C01800=1075.435,113.912,-70.031,173.707,24.375,154.288
C01801=1075.430,113.662,-70.011,173.705,24.372,154.287
C01802=1075.424,113.413,-69.992,173.704,24.370,154.287
C01803=1075.418,113.163,-69.973,173.702,24.367,154.287
C01804=1075.413,112.915,-69.954,173.700,24.364,154.287
C01805=1075.407,112.666,-69.935,173.699,24.362,154.286
C01806=1075.401,112.416,-69.916,173.697,24.360,154.286
C01807=1075.395,112.167,-69.896,173.695,24.357,154.286
C01808=1075.389,111.918,-69.877,173.694,24.355,154.285
C01809=1075.384,111.669,-69.858,173.693,24.352,154.285
C01810=1075.378,111.387,-69.837,173.690,24.349,154.285
C01811=1075.371,111.105,-69.815,173.688,24.346,154.284
C01812=1075.364,110.824,-69.794,173.687,24.343,154.284
C01813=1075.358,110.542,-69.773,173.684,24.341,154.284
C01814=1075.352,110.293,-69.754,173.683,24.338,154.283
C01815=1075.347,110.044,-69.734,173.681,24.335,154.283
C01816=1075.341,109.795,-69.716,173.680,24.333,154.283
C01817=1075.335,109.546,-69.697,173.678,24.330,154.283
C01818=1075.329,109.296,-69.678,173.676,24.328,154.282
C01819=1075.323,109.047,-69.659,173.675,24.325,154.282
C01820=1075.317,108.798,-69.640,173.673,24.323,154.282
C01821=1075.312,108.549,-69.621,173.671,24.320,154.282
C01822=1075.306,108.300,-69.602,173.670,24.318,154.281
C01823=1075.300,108.050,-69.583,173.668,24.316,154.281
C01824=1075.294,107.801,-69.564,173.666,24.313,154.281
C01825=1075.289,107.552,-69.545,173.665,24.311,154.280
C01826=1075.283,107.302,-69.527,173.663,24.308,154.280
C01827=1075.277,107.053,-69.508,173.661,24.305,154.280
C01828=1075.272,106.804,-69.489,173.660,24.303,154.279
C01829=1075.266,106.555,-69.470,173.658,24.300,154.279
C01830=1075.260,106.306,-69.451,173.656,24.298,154.279
C01831=1075.255,106.056,-69.432,173.655,24.295,154.279
C01832=1075.249,105.808,-69.413,173.653,24.293,154.278
C01833=1075.243,105.558,-69.395,173.651,24.290,154.278
C01834=1075.237,105.309,-69.376,173.650,24.287,154.278
C01835=1075.232,105.060,-69.357,173.649,24.285,154.277
C01836=1075.226,104.811,-69.338,173.646,24.282,154.277
C01837=1075.220,104.561,-69.320,173.645,24.280,154.277
C01838=1075.215,104.312,-69.301,173.644,24.277,154.277
C01839=1075.209,104.063,-69.282,173.642,24.275,154.276
C01840=1075.203,103.814,-69.263,173.640,24.272,154.276
C01841=1075.198,103.565,-69.244,173.639,24.269,154.276
C01842=1075.192,103.315,-69.226,173.637,24.267,154.275
C01843=1075.186,103.066,-69.207,173.635,24.264,154.275
C01844=1075.181,102.817,-69.188,173.634,24.262,154.275
C01845=1075.175,102.567,-69.170,173.632,24.260,154.274
C01846=1075.169,102.318,-69.151,173.630,24.256,154.274
C01847=1075.164,102.069,-69.132,173.629,24.254,154.274
C01848=1075.158,101.820,-69.114,173.627,24.252,154.274
C01849=1075.153,101.571,-69.096,173.625,24.249,154.273
C01850=1075.146,101.321,-69.077,173.624,24.247,154.273
C01851=1075.141,101.071,-69.058,173.623,24.244,154.273
C01852=1075.135,100.823,-69.040,173.621,24.241,154.272
C01853=1075.129,100.574,-69.021,173.619,24.239,154.272
C01854=1075.123,100.324,-69.003,173.618,24.236,154.272
C01855=1075.118,100.075,-68.984,173.616,24.234,154.271
C01856=1075.112,99.826,-68.965,173.614,24.231,154.271
C01857=1075.106,99.576,-68.947,173.613,24.229,154.271
C01858=1075.101,99.327,-68.929,173.611,24.227,154.271
C01859=1075.095,99.078,-68.911,173.609,24.224,154.270
C01860=1075.089,98.828,-68.891,173.608,24.221,154.270
C01861=1075.083,98.580,-68.873,173.606,24.219,154.270
C01862=1075.077,98.330,-68.855,173.605,24.216,154.269
C01863=1075.072,98.081,-68.836,173.603,24.213,154.269
C01864=1075.066,97.832,-68.818,173.602,24.211,154.269
C01865=1075.060,97.582,-68.799,173.600,24.209,154.269
C01866=1075.054,97.333,-68.782,173.598,24.206,154.268
C01867=1075.048,97.084,-68.763,173.597,24.203,154.268
C01868=1075.043,96.835,-68.745,173.595,24.201,154.268
C01869=1075.037,96.586,-68.726,173.593,24.198,154.267
C01870=1075.031,96.336,-68.708,173.592,24.196,154.267
C01871=1075.026,96.087,-68.689,173.590,24.193,154.267
C01872=1075.019,95.837,-68.671,173.589,24.191,154.266
C01873=1075.014,95.589,-68.652,173.587,24.188,154.266
C01874=1075.008,95.307,-68.632,173.586,24.185,154.266
C01875=1075.001,95.025,-68.612,173.583,24.182,154.265
C01876=1074.995,94.744,-68.591,173.582,24.180,154.265
C01877=1074.988,94.462,-68.570,173.580,24.176,154.265
C01878=1074.983,94.213,-68.551,173.579,24.174,154.264
C01879=1074.977,93.963,-68.533,173.576,24.171,154.264
C01880=1074.971,93.714,-68.516,173.575,24.168,154.264
C01881=1074.965,93.465,-68.497,173.574,24.166,154.263
C01882=1074.960,93.216,-68.479,173.572,24.164,154.263
C01883=1074.953,92.967,-68.460,173.570,24.161,154.263
C01884=1074.949,92.717,-68.442,173.569,24.159,154.263
C01885=1074.943,92.468,-68.424,173.568,24.156,154.262
C01886=1074.937,92.219,-68.406,173.566,24.153,154.262
C01887=1074.931,91.970,-68.388,173.564,24.151,154.262
C01888=1074.926,91.720,-68.370,173.563,24.148,154.261
C01889=1074.919,91.471,-68.351,173.561,24.145,154.261
C01890=1074.914,91.222,-68.334,173.559,24.143,154.261
C01891=1074.909,90.972,-68.315,173.558,24.140,154.260
C01892=1074.903,90.724,-68.297,173.556,24.138,154.260
C01893=1074.897,90.474,-68.279,173.555,24.136,154.260
C01894=1074.891,90.225,-68.261,173.553,24.132,154.259
C01895=1074.885,89.975,-68.243,173.552,24.130,154.259
C01896=1074.879,89.727,-68.225,173.550,24.128,154.259
C01897=1074.874,89.477,-68.207,173.549,24.125,154.259
C01898=1074.868,89.228,-68.189,173.547,24.122,154.258
C01899=1074.862,88.978,-68.171,173.545,24.120,154.258
C01900=1074.856,88.729,-68.153,173.544,24.117,154.258
C01901=1074.850,88.480,-68.135,173.543,24.115,154.257
C01902=1074.844,88.230,-68.117,173.541,24.112,154.257
C01903=1074.839,87.981,-68.099,173.539,24.110,154.257
C01904=1074.833,87.732,-68.081,173.538,24.107,154.257
C01905=1074.827,87.483,-68.063,173.537,24.105,154.256
C01906=1074.821,87.234,-68.046,173.534,24.102,154.256
C01907=1074.815,86.984,-68.028,173.533,24.099,154.256
C01908=1074.810,86.735,-68.010,173.532,24.097,154.255
C01909=1074.804,86.485,-67.992,173.530,24.095,154.255
C01910=1074.798,86.236,-67.973,173.528,24.092,154.255
C01911=1074.792,85.987,-67.955,173.527,24.089,154.254
C01912=1074.787,85.738,-67.938,173.526,24.087,154.254
C01913=1074.780,85.488,-67.920,173.524,24.084,154.254
C01914=1074.775,85.239,-67.902,173.522,24.081,154.254
C01915=1074.769,84.989,-67.884,173.521,24.079,154.253
C01916=1074.763,84.740,-67.867,173.519,24.076,154.253
C01917=1074.758,84.491,-67.849,173.518,24.074,154.253
C01918=1074.752,84.241,-67.831,173.516,24.071,154.252
C01919=1074.746,83.992,-67.814,173.514,24.069,154.252
C01920=1074.740,83.743,-67.795,173.513,24.066,154.252
C01921=1074.734,83.494,-67.778,173.512,24.063,154.251
C01922=1074.729,83.245,-67.760,173.510,24.061,154.251
C01923=1074.723,82.995,-67.742,173.508,24.058,154.251
C01924=1074.717,82.746,-67.725,173.507,24.056,154.250
C01925=1074.711,82.497,-67.707,173.506,24.053,154.250
C01926=1074.705,82.247,-67.689,173.504,24.050,154.250
C01927=1074.700,81.998,-67.671,173.502,24.048,154.249
C01928=1074.694,81.749,-67.654,173.501,24.046,154.249
C01929=1074.688,81.500,-67.636,173.500,24.043,154.249
C01930=1074.683,81.251,-67.618,173.497,24.040,154.249
C01931=1074.677,81.001,-67.600,173.496,24.038,154.248
C01932=1074.671,80.752,-67.583,173.495,24.035,154.248
C01933=1074.666,80.503,-67.565,173.494,24.032,154.248
C01934=1074.659,80.253,-67.547,173.491,24.030,154.247
C01935=1074.654,80.003,-67.531,173.490,24.027,154.247
C01936=1074.649,79.754,-67.513,173.489,24.024,154.247
C01937=1074.643,79.505,-67.495,173.487,24.022,154.246
C01938=1074.636,79.224,-67.475,173.485,24.019,154.246
C01939=1074.630,78.942,-67.455,173.484,24.016,154.246
C01940=1074.624,78.661,-67.435,173.482,24.013,154.245
C01941=1074.617,78.379,-67.415,173.481,24.010,154.245
C01942=1074.612,78.129,-67.398,173.478,24.007,154.245
C01943=1074.606,77.880,-67.380,173.477,24.005,154.244
C01944=1074.600,77.631,-67.363,173.476,24.003,154.244
C01945=1074.594,77.382,-67.346,173.475,24.000,154.244
C01946=1074.588,77.132,-67.328,173.472,23.997,154.243
C01947=1074.582,76.883,-67.310,173.471,23.994,154.243
C01948=1074.577,76.634,-67.292,173.470,23.992,154.243
C01949=1074.571,76.384,-67.275,173.469,23.989,154.242
C01950=1074.564,76.135,-67.258,173.467,23.987,154.242
C01951=1074.559,75.886,-67.241,173.465,23.984,154.242
C01952=1074.553,75.637,-67.223,173.464,23.982,154.242
C01953=1074.547,75.387,-67.205,173.462,23.979,154.241
C01954=1074.542,75.137,-67.188,173.461,23.976,154.241
C01955=1074.536,74.889,-67.171,173.459,23.974,154.241
C01956=1074.530,74.639,-67.153,173.457,23.971,154.240
C01957=1074.524,74.390,-67.136,173.456,23.969,154.240
C01958=1074.519,74.140,-67.119,173.455,23.966,154.240
C01959=1074.512,73.891,-67.102,173.454,23.964,154.239
C01960=1074.507,73.642,-67.084,173.451,23.961,154.239
C01961=1074.501,73.392,-67.067,173.450,23.958,154.239
C01962=1074.496,73.143,-67.050,173.449,23.956,154.238
C01963=1074.489,72.894,-67.032,173.448,23.953,154.238
C01964=1074.483,72.645,-67.015,173.446,23.951,154.238
C01965=1074.478,72.395,-66.998,173.444,23.948,154.237
C01966=1074.473,72.146,-66.980,173.443,23.945,154.237
C01967=1074.466,71.897,-66.963,173.441,23.943,154.237
C01968=1074.461,71.647,-66.946,173.440,23.940,154.237
C01969=1074.455,71.398,-66.929,173.438,23.937,154.236
C01970=1074.449,71.149,-66.912,173.437,23.935,154.236
C01971=1074.443,70.899,-66.894,173.435,23.932,154.236
C01972=1074.438,70.650,-66.877,173.434,23.930,154.235
C01973=1074.432,70.400,-66.860,173.433,23.927,154.235
C01974=1074.426,70.151,-66.843,173.431,23.924,154.235
C01975=1074.420,69.902,-66.825,173.429,23.922,154.234
C01976=1074.414,69.652,-66.809,173.428,23.919,154.234
C01977=1074.408,69.403,-66.791,173.427,23.917,154.234
C01978=1074.403,69.154,-66.774,173.425,23.914,154.233
C01979=1074.396,68.904,-66.757,173.423,23.911,154.233
C01980=1074.391,68.655,-66.740,173.422,23.909,154.233
C01981=1074.386,68.405,-66.723,173.421,23.906,154.232
C01982=1074.379,68.157,-66.706,173.419,23.904,154.232
C01983=1074.374,67.907,-66.689,173.418,23.901,154.232
C01984=1074.367,67.658,-66.672,173.416,23.898,154.231
C01985=1074.362,67.408,-66.655,173.415,23.896,154.231
C01986=1074.356,67.159,-66.638,173.413,23.893,154.231
C01987=1074.351,66.910,-66.621,173.412,23.891,154.231
C01988=1074.345,66.660,-66.603,173.411,23.888,154.230
C01989=1074.339,66.410,-66.587,173.408,23.885,154.230
C01990=1074.333,66.161,-66.569,173.407,23.883,154.230
C01991=1074.327,65.912,-66.553,173.406,23.881,154.229
C01992=1074.322,65.663,-66.535,173.405,23.878,154.229
C01993=1074.316,65.414,-66.519,173.403,23.875,154.229
C01994=1074.310,65.163,-66.502,173.401,23.872,154.228
C01995=1074.304,64.915,-66.485,173.400,23.870,154.228
C01996=1074.298,64.665,-66.468,173.399,23.867,154.228
C01997=1074.292,64.416,-66.451,173.397,23.865,154.227
C01998=1074.287,64.167,-66.434,173.396,23.862,154.227
C01999=1074.281,63.918,-66.417,173.394,23.860,154.227
C02000=1074.274,63.668,-66.401,173.392,23.857,154.226
C02001=1074.269,63.418,-66.384,173.391,23.854,154.226
C02002=1074.262,63.137,-66.365,173.389,23.852,154.226
C02003=1074.255,62.855,-66.346,173.388,23.849,154.226
C02004=1074.248,62.574,-66.327,173.386,23.846,154.225
C02005=1074.242,62.293,-66.308,173.384,23.843,154.225
C02006=1074.236,62.042,-66.291,173.383,23.841,154.225
C02007=1074.230,61.793,-66.274,173.382,23.838,154.224
C02008=1074.224,61.544,-66.258,173.380,23.835,154.224
C02009=1074.218,61.294,-66.241,173.378,23.833,154.224
C02010=1074.212,61.046,-66.224,173.377,23.830,154.223
C02011=1074.206,60.796,-66.208,173.376,23.828,154.223
C02012=1074.200,60.546,-66.191,173.374,23.825,154.223
C02013=1074.194,60.297,-66.174,173.373,23.822,154.222
C02014=1074.188,60.048,-66.157,173.371,23.820,154.222
C02015=1074.182,59.799,-66.141,173.370,23.817,154.222
C02016=1074.177,59.549,-66.124,173.368,23.815,154.222
C02017=1074.171,59.300,-66.107,173.367,23.812,154.221
C02018=1074.164,59.050,-66.091,173.366,23.810,154.221
C02019=1074.159,58.800,-66.074,173.364,23.807,154.221
C02020=1074.153,58.551,-66.058,173.362,23.804,154.220
C02021=1074.147,58.302,-66.041,173.361,23.802,154.220
C02022=1074.141,58.053,-66.024,173.360,23.799,154.220
C02023=1074.136,57.803,-66.008,173.358,23.797,154.219
C02024=1074.130,57.554,-65.991,173.357,23.794,154.219
C02025=1074.124,57.305,-65.975,173.355,23.792,154.219
C02026=1074.118,57.055,-65.959,173.354,23.789,154.218
C02027=1074.112,56.806,-65.941,173.352,23.786,154.218
C02028=1074.106,56.556,-65.925,173.351,23.784,154.218
C02029=1074.100,56.307,-65.908,173.350,23.781,154.217
C02030=1074.094,56.058,-65.892,173.348,23.778,154.217
C02031=1074.089,55.808,-65.875,173.346,23.776,154.217
C02032=1074.083,55.559,-65.859,173.345,23.773,154.217
C02033=1074.077,55.309,-65.843,173.344,23.771,154.216
C02034=1074.070,55.060,-65.826,173.342,23.768,154.216
C02035=1074.065,54.811,-65.809,173.341,23.766,154.216
C02036=1074.059,54.561,-65.793,173.339,23.763,154.215
C02037=1074.053,54.312,-65.776,173.338,23.761,154.215
C02038=1074.047,54.063,-65.760,173.336,23.758,154.215
C02039=1074.041,53.813,-65.744,173.335,23.755,154.214
C02040=1074.036,53.564,-65.727,173.334,23.753,154.214
C02041=1074.030,53.314,-65.711,173.333,23.750,154.214
C02042=1074.024,53.065,-65.695,173.330,23.747,154.213
C02043=1074.018,52.816,-65.678,173.329,23.745,154.213
C02044=1074.012,52.566,-65.662,173.328,23.742,154.213
C02045=1074.007,52.317,-65.645,173.327,23.739,154.212
C02046=1074.001,52.067,-65.629,173.325,23.737,154.212
C02047=1073.995,51.818,-65.613,173.323,23.734,154.212
C02048=1073.989,51.569,-65.596,173.322,23.731,154.211
C02049=1073.983,51.319,-65.580,173.321,23.729,154.211
C02050=1073.978,51.070,-65.563,173.319,23.727,154.211
C02051=1073.972,50.820,-65.547,173.318,23.724,154.210
C02052=1073.966,50.571,-65.531,173.317,23.721,154.210
C02053=1073.960,50.322,-65.515,173.315,23.718,154.210
C02054=1073.954,50.072,-65.498,173.313,23.716,154.210
C02055=1073.949,49.823,-65.481,173.312,23.713,154.209
C02056=1073.943,49.573,-65.465,173.311,23.711,154.209
C02057=1073.937,49.324,-65.449,173.309,23.708,154.209
C02058=1073.931,49.075,-65.433,173.308,23.705,154.208
C02059=1073.925,48.825,-65.416,173.306,23.703,154.208
C02060=1073.919,48.576,-65.400,173.305,23.700,154.208
C02061=1073.914,48.327,-65.384,173.304,23.697,154.207
C02062=1073.909,48.078,-65.367,173.302,23.695,154.207
C02063=1073.903,47.828,-65.352,173.301,23.693,154.207
C02064=1073.897,47.578,-65.336,173.300,23.690,154.206
C02065=1073.891,47.329,-65.319,173.298,23.687,154.206
C02066=1073.885,47.047,-65.301,173.296,23.684,154.206
C02067=1073.878,46.766,-65.283,173.295,23.681,154.205
C02068=1073.871,46.483,-65.264,173.293,23.678,154.205
C02069=1073.865,46.202,-65.246,173.292,23.675,154.205
C02070=1073.859,45.952,-65.230,173.291,23.673,154.204
C02071=1073.854,45.703,-65.213,173.288,23.669,154.204
C02072=1073.848,45.454,-65.197,173.287,23.667,154.204
C02073=1073.843,45.204,-65.182,173.286,23.664,154.203
C02074=1073.837,44.955,-65.165,173.285,23.662,154.203
C02075=1073.831,44.705,-65.149,173.283,23.659,154.203
C02076=1073.825,44.456,-65.133,173.282,23.656,154.202
C02077=1073.819,44.206,-65.117,173.280,23.654,154.202
C02078=1073.813,43.957,-65.101,173.279,23.651,154.202
C02079=1073.808,43.708,-65.085,173.278,23.648,154.201
C02080=1073.802,43.459,-65.069,173.276,23.646,154.201
C02081=1073.796,43.209,-65.053,173.275,23.644,154.201
C02082=1073.790,42.959,-65.037,173.274,23.641,154.200
C02083=1073.785,42.710,-65.021,173.272,23.638,154.200
C02084=1073.779,42.461,-65.005,173.270,23.635,154.200
C02085=1073.773,42.211,-64.989,173.269,23.633,154.199
C02086=1073.767,41.961,-64.973,173.268,23.631,154.199
C02087=1073.761,41.712,-64.957,173.266,23.628,154.199
C02088=1073.756,41.463,-64.941,173.265,23.625,154.198
C02089=1073.750,41.213,-64.925,173.264,23.623,154.198
C02090=1073.743,40.964,-64.910,173.262,23.620,154.198
C02091=1073.738,40.714,-64.894,173.260,23.617,154.198
C02092=1073.732,40.465,-64.878,173.259,23.615,154.197
C02093=1073.726,40.216,-64.861,173.258,23.612,154.197
C02094=1073.721,39.966,-64.846,173.257,23.609,154.197
C02095=1073.715,39.717,-64.830,173.255,23.607,154.196
C02096=1073.709,39.467,-64.814,173.254,23.605,154.196
C02097=1073.703,39.218,-64.798,173.252,23.601,154.196
C02098=1073.697,38.968,-64.782,173.251,23.599,154.195
C02099=1073.691,38.719,-64.767,173.249,23.596,154.195
C02100=1073.686,38.470,-64.751,173.248,23.594,154.195
C02101=1073.680,38.220,-64.736,173.247,23.591,154.194
C02102=1073.674,37.971,-64.719,173.246,23.589,154.194
C02103=1073.668,37.721,-64.703,173.244,23.586,154.194
C02104=1073.662,37.471,-64.688,173.242,23.584,154.194
C02105=1073.656,37.222,-64.672,173.241,23.581,154.193
C02106=1073.651,36.973,-64.657,173.240,23.578,154.193
C02107=1073.645,36.724,-64.640,173.238,23.576,154.193
C02108=1073.638,36.474,-64.625,173.237,23.573,154.192
C02109=1073.632,36.225,-64.609,173.236,23.570,154.192
C02110=1073.627,35.975,-64.594,173.234,23.568,154.192
C02111=1073.621,35.726,-64.578,173.232,23.565,154.191
C02112=1073.615,35.476,-64.563,173.231,23.563,154.191
C02113=1073.609,35.227,-64.547,173.230,23.560,154.191
C02114=1073.603,34.977,-64.531,173.229,23.558,154.190
C02115=1073.597,34.728,-64.515,173.227,23.555,154.190
C02116=1073.592,34.479,-64.500,173.226,23.553,154.190
C02117=1073.586,34.229,-64.484,173.224,23.550,154.189
C02118=1073.579,33.980,-64.469,173.222,23.548,154.189
C02119=1073.574,33.730,-64.453,173.221,23.545,154.189
C02120=1073.568,33.480,-64.437,173.220,23.542,154.189
C02121=1073.562,33.232,-64.423,173.219,23.540,154.188
C02122=1073.556,32.982,-64.406,173.217,23.537,154.188
C02123=1073.550,32.732,-64.391,173.216,23.534,154.188
C02124=1073.544,32.483,-64.376,173.214,23.532,154.187
C02125=1073.539,32.234,-64.360,173.213,23.529,154.187
C02126=1073.533,31.984,-64.344,173.211,23.527,154.187
C02127=1073.526,31.735,-64.329,173.210,23.524,154.186
C02128=1073.521,31.485,-64.313,173.209,23.521,154.186
C02129=1073.516,31.236,-64.298,173.208,23.519,154.186
C02130=1073.508,30.954,-64.281,173.206,23.516,154.185
C02131=1073.502,30.672,-64.263,173.204,23.513,154.185
C02132=1073.495,30.390,-64.246,173.203,23.510,154.185
C02133=1073.489,30.108,-64.228,173.201,23.507,154.184
C02134=1073.483,29.859,-64.213,173.200,23.505,154.184
C02135=1073.477,29.609,-64.197,173.199,23.502,154.184
C02136=1073.471,29.360,-64.182,173.197,23.499,154.183
C02137=1073.465,29.110,-64.167,173.196,23.497,154.183
C02138=1073.459,28.861,-64.150,173.194,23.494,154.183
C02139=1073.453,28.612,-64.136,173.193,23.492,154.182
C02140=1073.448,28.362,-64.120,173.191,23.489,154.182
C02141=1073.441,28.112,-64.105,173.190,23.486,154.182
C02142=1073.436,27.864,-64.089,173.189,23.484,154.182
C02143=1073.430,27.614,-64.074,173.188,23.482,154.181
C02144=1073.424,27.364,-64.059,173.186,23.479,154.181
C02145=1073.418,27.115,-64.044,173.185,23.477,154.181
C02146=1073.413,26.865,-64.029,173.183,23.473,154.180
C02147=1073.406,26.616,-64.013,173.182,23.471,154.180
C02148=1073.400,26.366,-63.998,173.180,23.469,154.180
C02149=1073.394,26.117,-63.983,173.179,23.466,154.179
C02150=1073.389,25.867,-63.967,173.178,23.464,154.179
C02151=1073.382,25.618,-63.953,173.176,23.461,154.179
C02152=1073.376,25.369,-63.937,173.175,23.458,154.178
C02153=1073.371,25.119,-63.922,173.173,23.456,154.178
C02154=1073.364,24.870,-63.907,173.172,23.453,154.178
C02155=1073.359,24.620,-63.892,173.170,23.451,154.178
C02156=1073.353,24.371,-63.877,173.169,23.448,154.177
C02157=1073.347,24.121,-63.861,173.168,23.445,154.177
C02158=1073.342,23.872,-63.847,173.167,23.443,154.177
C02159=1073.335,23.623,-63.831,173.165,23.441,154.176
C02160=1073.329,23.373,-63.815,173.164,23.438,154.176
C02161=1073.323,23.124,-63.801,173.162,23.435,154.176
C02162=1073.318,22.874,-63.785,173.161,23.433,154.176
C02163=1073.311,22.624,-63.770,173.159,23.430,154.175
C02164=1073.306,22.375,-63.755,173.158,23.428,154.175
C02165=1073.300,22.125,-63.740,173.157,23.425,154.175
C02166=1073.294,21.876,-63.726,173.156,23.423,154.174
C02167=1073.289,21.626,-63.710,173.154,23.420,154.174
C02168=1073.282,21.377,-63.695,173.153,23.417,154.174
C02169=1073.277,21.128,-63.680,173.151,23.415,154.173
C02170=1073.271,20.878,-63.665,173.150,23.412,154.173
C02171=1073.264,20.628,-63.650,173.148,23.410,154.173
C02172=1073.259,20.379,-63.635,173.147,23.407,154.172
C02173=1073.253,20.129,-63.620,173.146,23.404,154.172
C02174=1073.247,19.880,-63.605,173.145,23.402,154.172
C02175=1073.241,19.630,-63.590,173.143,23.400,154.172
C02176=1073.235,19.381,-63.575,173.142,23.397,154.171
C02177=1073.229,19.132,-63.560,173.140,23.394,154.171
C02178=1073.223,18.882,-63.545,173.138,23.392,154.171
C02179=1073.218,18.633,-63.530,173.137,23.390,154.170
C02180=1073.211,18.383,-63.515,173.136,23.387,154.170
C02181=1073.205,18.134,-63.500,173.135,23.384,154.170
C02182=1073.200,17.884,-63.485,173.133,23.382,154.169
C02183=1073.194,17.635,-63.470,173.132,23.379,154.169
C02184=1073.188,17.386,-63.456,173.131,23.377,154.169
C02185=1073.182,17.136,-63.441,173.129,23.374,154.169
C02186=1073.176,16.887,-63.425,173.127,23.372,154.168
C02187=1073.170,16.637,-63.410,173.126,23.369,154.168
C02188=1073.165,16.387,-63.397,173.125,23.366,154.168
C02189=1073.158,16.138,-63.382,173.124,23.364,154.167
C02190=1073.153,15.888,-63.366,173.122,23.362,154.167
C02191=1073.147,15.639,-63.352,173.121,23.359,154.167
C02192=1073.140,15.389,-63.337,173.120,23.357,154.167
C02193=1073.135,15.140,-63.322,173.118,23.353,154.166
C02194=1073.128,14.860,-63.305,173.116,23.351,154.166
C02195=1073.121,14.580,-63.289,173.115,23.348,154.165
C02196=1073.115,14.299,-63.272,173.113,23.345,154.165
C02197=1073.108,14.018,-63.255,173.112,23.342,154.165
C02198=1073.102,13.769,-63.241,173.111,23.340,154.165
C02199=1073.096,13.519,-63.227,173.109,23.337,154.164
C02200=1073.090,13.270,-63.212,173.108,23.335,154.164
C02201=1073.084,13.021,-63.197,173.106,23.332,154.164
C02202=1073.078,12.770,-63.182,173.105,23.330,154.163
C02203=1073.073,12.521,-63.168,173.103,23.327,154.163
C02204=1073.066,12.271,-63.153,173.102,23.325,154.163
C02205=1073.060,12.022,-63.138,173.101,23.323,154.163
C02206=1073.054,11.772,-63.124,173.099,23.320,154.162
C02207=1073.049,11.523,-63.109,173.098,23.318,154.162
C02208=1073.042,11.274,-63.094,173.097,23.315,154.162
C02209=1073.036,11.025,-63.080,173.096,23.313,154.161
C02210=1073.030,10.774,-63.066,173.093,23.310,154.161
C02211=1073.025,10.525,-63.051,173.092,23.308,154.161
C02212=1073.018,10.276,-63.036,173.091,23.305,154.161
C02213=1073.013,10.026,-63.022,173.090,23.303,154.160
C02214=1073.006,9.776,-63.007,173.088,23.300,154.160
C02215=1073.001,9.528,-62.993,173.087,23.298,154.160
C02216=1072.994,9.277,-62.978,173.086,23.296,154.159
C02217=1072.989,9.028,-62.964,173.084,23.293,154.159
C02218=1072.982,8.779,-62.949,173.082,23.290,154.159
C02219=1072.977,8.529,-62.935,173.081,23.287,154.159
C02220=1072.970,8.279,-62.920,173.080,23.285,154.158
C02221=1072.965,8.030,-62.905,173.078,23.283,154.158
C02222=1072.959,7.780,-62.891,173.077,23.280,154.158
C02223=1072.953,7.531,-62.877,173.076,23.278,154.157
C02224=1072.946,7.282,-62.862,173.075,23.275,154.157
C02225=1072.941,7.032,-62.848,173.073,23.273,154.157
C02226=1072.935,6.782,-62.833,173.072,23.270,154.157
C02227=1072.929,6.533,-62.819,173.070,23.268,154.156
C02228=1072.923,6.283,-62.804,173.069,23.265,154.156
C02229=1072.917,6.034,-62.790,173.067,23.263,154.156
C02230=1072.911,5.785,-62.776,173.066,23.260,154.155
C02231=1072.905,5.535,-62.761,173.065,23.258,154.155
C02232=1072.900,5.285,-62.747,173.063,23.255,154.155
C02233=1072.893,5.036,-62.732,173.062,23.253,154.155
C02234=1072.888,4.786,-62.718,173.061,23.251,154.154
C02235=1072.881,4.537,-62.704,173.059,23.248,154.154
C02236=1072.875,4.287,-62.690,173.057,23.245,154.154
C02237=1072.869,4.038,-62.675,173.056,23.242,154.153
C02238=1072.863,3.788,-62.661,173.055,23.240,154.153
C02239=1072.857,3.539,-62.646,173.054,23.238,154.153
C02240=1072.852,3.289,-62.633,173.052,23.235,154.153
C02241=1072.846,3.040,-62.618,173.051,23.233,154.152
C02242=1072.840,2.790,-62.604,173.050,23.230,154.152
C02243=1072.834,2.541,-62.589,173.049,23.228,154.152
C02244=1072.828,2.291,-62.575,173.046,23.225,154.151
C02245=1072.823,2.041,-62.561,173.045,23.223,154.151
C02246=1072.816,1.792,-62.546,173.044,23.220,154.151
C02247=1072.811,1.542,-62.532,173.042,23.218,154.151
C02248=1072.805,1.293,-62.518,173.041,23.215,154.150
C02249=1072.798,1.043,-62.504,173.040,23.213,154.150
C02250=1072.793,0.794,-62.489,173.039,23.211,154.150
C02251=1072.787,0.545,-62.476,173.037,23.208,154.149
C02252=1072.781,0.294,-62.461,173.036,23.206,154.149
C02253=1072.775,0.045,-62.447,173.034,23.203,154.149
C02254=1072.770,-0.204,-62.433,173.033,23.200,154.149
C02255=1072.764,-0.454,-62.419,173.031,23.198,154.148
C02256=1072.758,-0.703,-62.404,173.030,23.196,154.148
C02257=1072.752,-0.953,-62.390,173.029,23.193,154.148
C02258=1072.745,-1.231,-62.374,173.028,23.190,154.147
C02259=1072.739,-1.510,-62.359,173.025,23.187,154.147
C02260=1072.732,-1.788,-62.343,173.024,23.184,154.147
C02261=1072.726,-2.067,-62.327,173.023,23.182,154.146
C02262=1072.720,-2.316,-62.313,173.021,23.179,154.146
C02263=1072.714,-2.565,-62.299,173.020,23.177,154.146
C02264=1072.709,-2.815,-62.285,173.018,23.174,154.146
C02265=1072.702,-3.065,-62.270,173.017,23.172,154.145
C02266=1072.697,-3.314,-62.257,173.016,23.170,154.145
C02267=1072.691,-3.564,-62.243,173.014,23.167,154.145
C02268=1072.685,-3.814,-62.229,173.013,23.165,154.145
C02269=1072.679,-4.063,-62.215,173.012,23.162,154.144
C02270=1072.673,-4.312,-62.201,173.011,23.160,154.144
C02271=1072.667,-4.562,-62.187,173.009,23.157,154.144
C02272=1072.661,-4.812,-62.173,173.007,23.155,154.143
C02273=1072.655,-5.061,-62.159,173.006,23.152,154.143
C02274=1072.648,-5.311,-62.145,173.004,23.150,154.143
C02275=1072.643,-5.560,-62.131,173.003,23.148,154.143
C02276=1072.637,-5.810,-62.118,173.002,23.145,154.142
C02277=1072.631,-6.060,-62.104,173.001,23.143,154.142
C02278=1072.625,-6.309,-62.089,172.999,23.141,154.142
C02279=1072.619,-6.558,-62.076,172.998,23.138,154.142
C02280=1072.613,-6.808,-62.062,172.997,23.136,154.141
C02281=1072.606,-7.058,-62.048,172.995,23.133,154.141
C02282=1072.601,-7.307,-62.034,172.993,23.130,154.141
C02283=1072.595,-7.557,-62.020,172.992,23.129,154.141
C02284=1072.588,-7.806,-62.006,172.991,23.126,154.140
C02285=1072.583,-8.056,-61.992,172.989,23.124,154.140
C02286=1072.577,-8.305,-61.979,172.988,23.121,154.140
C02287=1072.571,-8.555,-61.965,172.987,23.119,154.140
C02288=1072.565,-8.805,-61.951,172.985,23.116,154.139
C02289=1072.559,-9.054,-61.938,172.984,23.114,154.139
C02290=1072.553,-9.304,-61.924,172.982,23.111,154.139
C02291=1072.547,-9.553,-61.911,172.981,23.109,154.138
C02292=1072.541,-9.803,-61.896,172.979,23.107,154.138
C02293=1072.535,-10.053,-61.883,172.978,23.104,154.138
C02294=1072.529,-10.302,-61.869,172.977,23.102,154.138
C02295=1072.524,-10.551,-61.855,172.975,23.100,154.137
C02296=1072.517,-10.800,-61.841,172.974,23.097,154.137
C02297=1072.511,-11.051,-61.827,172.973,23.095,154.137
C02298=1072.505,-11.300,-61.814,172.972,23.092,154.137
C02299=1072.500,-11.549,-61.800,172.969,23.089,154.136
C02300=1072.493,-11.799,-61.787,172.968,23.088,154.136
C02301=1072.488,-12.048,-61.773,172.967,23.085,154.136
C02302=1072.481,-12.298,-61.759,172.965,23.083,154.136
C02303=1072.476,-12.548,-61.745,172.964,23.080,154.135
C02304=1072.470,-12.797,-61.731,172.963,23.078,154.135
C02305=1072.464,-13.047,-61.718,172.962,23.075,154.135
C02306=1072.458,-13.296,-61.704,172.960,23.073,154.135
C02307=1072.452,-13.545,-61.691,172.959,23.071,154.134
C02308=1072.446,-13.796,-61.677,172.958,23.069,154.134
C02309=1072.440,-14.045,-61.664,172.955,23.066,154.134
C02310=1072.435,-14.295,-61.650,172.954,23.063,154.134
C02311=1072.429,-14.544,-61.637,172.953,23.061,154.133
C02312=1072.423,-14.794,-61.623,172.952,23.059,154.133
C02313=1072.417,-15.043,-61.610,172.950,23.056,154.133
C02314=1072.411,-15.293,-61.596,172.949,23.054,154.133
C02315=1072.405,-15.543,-61.582,172.948,23.052,154.132
C02316=1072.398,-15.792,-61.569,172.946,23.049,154.132
C02317=1072.393,-16.042,-61.555,172.945,23.047,154.132
C02318=1072.387,-16.291,-61.542,172.944,23.045,154.132
C02319=1072.380,-16.540,-61.529,172.941,23.042,154.131
C02320=1072.374,-16.791,-61.515,172.940,23.040,154.131
C02321=1072.369,-17.040,-61.502,172.939,23.037,154.131
C02322=1072.362,-17.317,-61.488,172.938,23.035,154.130
C02323=1072.355,-17.594,-61.472,172.936,23.032,154.130
C02324=1072.349,-17.871,-61.458,172.934,23.030,154.130
C02325=1072.342,-18.148,-61.443,172.933,23.027,154.130
C02326=1072.336,-18.397,-61.429,172.932,23.025,154.130
C02327=1072.330,-18.646,-61.416,172.930,23.023,154.129
C02328=1072.324,-18.896,-61.402,172.929,23.020,154.129
C02329=1072.318,-19.145,-61.388,172.927,23.018,154.129
C02330=1072.312,-19.395,-61.376,172.925,23.016,154.129
C02331=1072.306,-19.644,-61.363,172.924,23.013,154.128
C02332=1072.301,-19.894,-61.349,172.923,23.011,154.128
C02333=1072.294,-20.144,-61.335,172.922,23.008,154.128
C02334=1072.288,-20.394,-61.322,172.920,23.007,154.128
C02335=1072.282,-20.643,-61.309,172.919,23.004,154.127
C02336=1072.276,-20.893,-61.295,172.918,23.002,154.127
C02337=1072.270,-21.142,-61.282,172.916,23.000,154.127
C02338=1072.264,-21.392,-61.270,172.915,22.997,154.127
C02339=1072.259,-21.641,-61.256,172.913,22.995,154.126
C02340=1072.252,-21.891,-61.242,172.911,22.992,154.126
C02341=1072.246,-22.141,-61.230,172.910,22.990,154.126
C02342=1072.240,-22.390,-61.217,172.909,22.988,154.126
C02343=1072.235,-22.639,-61.203,172.907,22.985,154.125
C02344=1072.229,-22.889,-61.189,172.906,22.983,154.125
C02345=1072.222,-23.139,-61.177,172.905,22.981,154.125
C02346=1072.216,-23.389,-61.163,172.903,22.979,154.125
C02347=1072.210,-23.638,-61.149,172.902,22.976,154.124
C02348=1072.204,-23.888,-61.137,172.901,22.974,154.124
C02349=1072.198,-24.137,-61.124,172.899,22.971,154.124
C02350=1072.192,-24.387,-61.111,172.897,22.969,154.124
C02351=1072.187,-24.637,-61.097,172.896,22.967,154.124
C02352=1072.181,-24.886,-61.084,172.895,22.965,154.123
C02353=1072.175,-25.136,-61.071,172.893,22.962,154.123
C02354=1072.168,-25.385,-61.058,172.892,22.960,154.123
C02355=1072.163,-25.635,-61.044,172.891,22.958,154.123
C02356=1072.157,-25.885,-61.032,172.889,22.955,154.122
C02357=1072.151,-26.134,-61.018,172.888,22.954,154.122
C02358=1072.145,-26.384,-61.006,172.887,22.951,154.122
C02359=1072.140,-26.633,-60.992,172.884,22.948,154.122
C02360=1072.134,-26.883,-60.979,172.883,22.946,154.121
C02361=1072.127,-27.132,-60.966,172.882,22.944,154.121
C02362=1072.121,-27.382,-60.953,172.881,22.942,154.121
C02363=1072.115,-27.632,-60.940,172.879,22.940,154.121
C02364=1072.109,-27.881,-60.927,172.878,22.937,154.120
C02365=1072.103,-28.131,-60.914,172.876,22.935,154.120
C02366=1072.097,-28.380,-60.901,172.875,22.933,154.120
C02367=1072.091,-28.630,-60.889,172.874,22.931,154.120
C02368=1072.085,-28.879,-60.875,172.872,22.929,154.120
C02369=1072.079,-29.129,-60.863,172.870,22.926,154.119
C02370=1072.073,-29.378,-60.850,172.869,22.924,154.119
C02371=1072.067,-29.628,-60.837,172.868,22.921,154.119
C02372=1072.061,-29.877,-60.824,172.866,22.920,154.119
C02373=1072.055,-30.127,-60.811,172.865,22.917,154.118
C02374=1072.048,-30.377,-60.798,172.863,22.915,154.118
C02375=1072.043,-30.626,-60.785,172.862,22.913,154.118
C02376=1072.037,-30.876,-60.773,172.861,22.911,154.118
C02377=1072.030,-31.126,-60.760,172.859,22.908,154.118
C02378=1072.024,-31.376,-60.747,172.858,22.907,154.117
C02379=1072.018,-31.625,-60.734,172.857,22.904,154.117
C02380=1072.012,-31.875,-60.721,172.854,22.902,154.117
C02381=1072.006,-32.124,-60.708,172.853,22.899,154.117
C02382=1072.000,-32.374,-60.695,172.852,22.897,154.117
C02383=1071.994,-32.624,-60.683,172.850,22.895,154.116
C02384=1071.988,-32.873,-60.670,172.849,22.893,154.116
C02385=1071.982,-33.123,-60.657,172.848,22.891,154.116
C02386=1071.976,-33.399,-60.643,172.846,22.888,154.116
C02387=1071.970,-33.675,-60.628,172.844,22.885,154.115
C02388=1071.963,-33.950,-60.615,172.843,22.884,154.115
C02389=1071.956,-34.227,-60.600,172.842,22.881,154.115
C02390=1071.950,-34.476,-60.588,172.840,22.879,154.115
C02391=1071.944,-34.726,-60.575,172.839,22.877,154.115
C02392=1071.938,-34.976,-60.562,172.837,22.874,154.114
C02393=1071.932,-35.226,-60.549,172.835,22.872,154.114
C02394=1071.926,-35.475,-60.537,172.834,22.870,154.114
C02395=1071.921,-35.724,-60.524,172.833,22.868,154.114
C02396=1071.915,-35.974,-60.511,172.831,22.865,154.113
C02397=1071.909,-36.224,-60.499,172.830,22.863,154.113
C02398=1071.903,-36.473,-60.485,172.829,22.861,154.113
C02399=1071.897,-36.723,-60.473,172.827,22.859,154.113
C02400=1071.890,-36.972,-60.461,172.826,22.857,154.113
C02401=1071.884,-37.222,-60.448,172.824,22.855,154.112
C02402=1071.879,-37.471,-60.436,172.823,22.852,154.112
C02403=1071.873,-37.721,-60.423,172.821,22.850,154.112
C02404=1071.867,-37.971,-60.410,172.819,22.848,154.112
C02405=1071.861,-38.221,-60.398,172.818,22.846,154.112
C02406=1071.855,-38.470,-60.385,172.817,22.844,154.111
C02407=1071.849,-38.720,-60.372,172.816,22.841,154.111
C02408=1071.843,-38.970,-60.359,172.814,22.839,154.111
C02409=1071.836,-39.219,-60.348,172.813,22.837,154.111
C02410=1071.831,-39.468,-60.335,172.811,22.835,154.111
C02411=1071.825,-39.718,-60.323,172.810,22.833,154.110
C02412=1071.819,-39.967,-60.309,172.809,22.831,154.110
C02413=1071.812,-40.217,-60.298,172.807,22.829,154.110
C02414=1071.806,-40.467,-60.285,172.805,22.826,154.110
C02415=1071.800,-40.717,-60.272,172.804,22.824,154.110
C02416=1071.794,-40.967,-60.260,172.802,22.822,154.109
C02417=1071.788,-41.216,-60.248,172.801,22.820,154.109
C02418=1071.782,-41.465,-60.236,172.800,22.818,154.109
C02419=1071.776,-41.715,-60.222,172.798,22.816,154.109
C02420=1071.770,-41.965,-60.210,172.797,22.814,154.109
C02421=1071.764,-42.214,-60.198,172.795,22.812,154.108
C02422=1071.758,-42.464,-60.185,172.794,22.810,154.108
C02423=1071.752,-42.714,-60.173,172.793,22.808,154.108
C02424=1071.747,-42.963,-60.161,172.791,22.805,154.108
C02425=1071.740,-43.213,-60.149,172.789,22.803,154.108
C02426=1071.734,-43.463,-60.136,172.788,22.801,154.108
C02427=1071.728,-43.712,-60.124,172.786,22.799,154.107
C02428=1071.721,-43.962,-60.112,172.785,22.797,154.107
C02429=1071.716,-44.211,-60.099,172.783,22.795,154.107
C02430=1071.710,-44.461,-60.087,172.782,22.793,154.107
C02431=1071.704,-44.711,-60.075,172.781,22.791,154.107
C02432=1071.698,-44.961,-60.062,172.779,22.789,154.106
C02433=1071.692,-45.210,-60.050,172.778,22.787,154.106
C02434=1071.686,-45.460,-60.038,172.776,22.785,154.106
C02435=1071.680,-45.709,-60.026,172.775,22.782,154.106
C02436=1071.674,-45.959,-60.013,172.774,22.781,154.106
C02437=1071.668,-46.209,-60.001,172.771,22.778,154.106
C02438=1071.662,-46.458,-59.989,172.770,22.776,154.105
C02439=1071.656,-46.708,-59.976,172.769,22.774,154.105
C02440=1071.650,-46.958,-59.964,172.767,22.772,154.105
C02441=1071.644,-47.207,-59.952,172.766,22.770,154.105
C02442=1071.638,-47.456,-59.940,172.765,22.768,154.105
C02443=1071.632,-47.706,-59.927,172.763,22.766,154.104
C02444=1071.626,-47.956,-59.915,172.762,22.764,154.104
C02445=1071.620,-48.206,-59.903,172.760,22.762,154.104
C02446=1071.614,-48.455,-59.890,172.759,22.759,154.104
C02447=1071.608,-48.704,-59.879,172.758,22.758,154.104
C02448=1071.602,-48.954,-59.866,172.756,22.756,154.104
C02449=1071.597,-49.203,-59.854,172.755,22.754,154.103
C02450=1071.590,-49.480,-59.841,172.753,22.751,154.103
C02451=1071.582,-49.757,-59.827,172.751,22.749,154.103
C02452=1071.577,-50.033,-59.814,172.750,22.747,154.103
C02453=1071.570,-50.310,-59.801,172.748,22.744,154.103
C02454=1071.564,-50.560,-59.788,172.746,22.742,154.103
C02455=1071.558,-50.809,-59.777,172.745,22.741,154.102
C02456=1071.551,-51.058,-59.765,172.743,22.739,154.102
C02457=1071.545,-51.308,-59.752,172.742,22.736,154.102
C02458=1071.539,-51.558,-59.740,172.741,22.734,154.102
C02459=1071.533,-51.808,-59.728,172.739,22.732,154.102
C02460=1071.527,-52.057,-59.717,172.738,22.730,154.102
C02461=1071.520,-52.307,-59.705,172.736,22.729,154.101
C02462=1071.514,-52.556,-59.692,172.735,22.727,154.101
C02463=1071.508,-52.806,-59.680,172.733,22.725,154.101
C02464=1071.502,-53.056,-59.669,172.731,22.722,154.101
C02465=1071.496,-53.305,-59.657,172.730,22.721,154.101
C02466=1071.489,-53.555,-59.645,172.728,22.719,154.101
C02467=1071.483,-53.804,-59.633,172.727,22.717,154.101
C02468=1071.478,-54.054,-59.621,172.725,22.715,154.100
C02469=1071.471,-54.304,-59.609,172.724,22.713,154.100
C02470=1071.464,-54.553,-59.597,172.723,22.711,154.100
C02471=1071.459,-54.803,-59.585,172.721,22.709,154.100
C02472=1071.453,-55.053,-59.574,172.720,22.707,154.100
C02473=1071.446,-55.302,-59.562,172.718,22.705,154.100
C02474=1071.441,-55.552,-59.550,172.717,22.703,154.099
C02475=1071.434,-55.801,-59.538,172.715,22.702,154.099
C02476=1071.428,-56.051,-59.527,172.714,22.700,154.099
C02477=1071.422,-56.301,-59.514,172.713,22.698,154.099
C02478=1071.416,-56.550,-59.503,172.710,22.695,154.099
C02479=1071.410,-56.800,-59.491,172.709,22.694,154.099
C02480=1071.404,-57.050,-59.479,172.707,22.692,154.099
C02481=1071.398,-57.299,-59.467,172.706,22.690,154.098
C02482=1071.391,-57.549,-59.456,172.704,22.688,154.098
C02483=1071.385,-57.799,-59.443,172.703,22.686,154.098
C02484=1071.379,-58.048,-59.432,172.702,22.684,154.098
C02485=1071.373,-58.298,-59.421,172.700,22.682,154.098
C02486=1071.368,-58.547,-59.408,172.699,22.680,154.098
C02487=1071.361,-58.798,-59.397,172.697,22.678,154.098
C02488=1071.355,-59.047,-59.385,172.696,22.676,154.097
C02489=1071.349,-59.296,-59.374,172.694,22.675,154.097
C02490=1071.343,-59.547,-59.362,172.693,22.673,154.097
C02491=1071.336,-59.796,-59.350,172.691,22.671,154.097
C02492=1071.331,-60.046,-59.339,172.690,22.669,154.097
C02493=1071.325,-60.295,-59.326,172.688,22.667,154.097
C02494=1071.319,-60.544,-59.315,172.686,22.665,154.097
C02495=1071.312,-60.795,-59.303,172.685,22.663,154.097
C02496=1071.306,-61.044,-59.291,172.683,22.661,154.096
C02497=1071.301,-61.294,-59.280,172.682,22.660,154.096
C02498=1071.294,-61.543,-59.268,172.681,22.658,154.096
C02499=1071.288,-61.793,-59.257,172.679,22.656,154.096
C02500=1071.282,-62.043,-59.245,172.678,22.654,154.096
C02501=1071.277,-62.292,-59.234,172.676,22.652,154.096
C02502=1071.270,-62.542,-59.222,172.675,22.651,154.096
C02503=1071.264,-62.792,-59.211,172.673,22.649,154.095
C02504=1071.258,-63.041,-59.198,172.672,22.647,154.095
C02505=1071.252,-63.291,-59.187,172.670,22.645,154.095
C02506=1071.246,-63.540,-59.176,172.669,22.643,154.095
C02507=1071.240,-63.791,-59.164,172.668,22.641,154.095
C02508=1071.234,-64.040,-59.152,172.666,22.639,154.095
C02509=1071.228,-64.290,-59.141,172.664,22.637,154.095
C02510=1071.222,-64.539,-59.129,172.662,22.635,154.095
C02511=1071.216,-64.789,-59.118,172.661,22.634,154.094
C02512=1071.210,-65.038,-59.107,172.659,22.632,154.094
C02513=1071.204,-65.288,-59.095,172.658,22.630,154.094
C02514=1071.197,-65.566,-59.082,172.656,22.628,154.094
C02515=1071.190,-65.844,-59.069,172.655,22.626,154.094
C02516=1071.184,-66.121,-59.056,172.653,22.624,154.094
C02517=1071.177,-66.399,-59.044,172.651,22.622,154.094
C02518=1071.171,-66.649,-59.032,172.650,22.620,154.093
C02519=1071.165,-66.898,-59.022,172.648,22.618,154.093
C02520=1071.159,-67.148,-59.009,172.647,22.616,154.093
C02521=1071.153,-67.398,-58.998,172.646,22.614,154.093
C02522=1071.147,-67.648,-58.987,172.644,22.613,154.093
C02523=1071.141,-67.897,-58.975,172.643,22.611,154.093
C02524=1071.135,-68.147,-58.964,172.641,22.609,154.093
C02525=1071.130,-68.397,-58.953,172.640,22.607,154.093
C02526=1071.123,-68.646,-58.941,172.638,22.605,154.092
C02527=1071.117,-68.896,-58.930,172.637,22.604,154.092
C02528=1071.111,-69.146,-58.918,172.634,22.602,154.092
C02529=1071.105,-69.395,-58.907,172.633,22.600,154.092
C02530=1071.100,-69.645,-58.895,172.631,22.598,154.092
C02531=1071.094,-69.895,-58.884,172.630,22.596,154.092
C02532=1071.088,-70.144,-58.873,172.628,22.594,154.092
C02533=1071.081,-70.394,-58.861,172.627,22.593,154.092
C02534=1071.075,-70.643,-58.850,172.626,22.591,154.092
C02535=1071.069,-70.894,-58.839,172.624,22.589,154.091
C02536=1071.064,-71.143,-58.827,172.623,22.587,154.091
C02537=1071.058,-71.392,-58.816,172.621,22.585,154.091
C02538=1071.052,-71.642,-58.805,172.620,22.584,154.091
C02539=1071.046,-71.892,-58.794,172.618,22.582,154.091
C02540=1071.039,-72.142,-58.782,172.617,22.580,154.091
C02541=1071.034,-72.391,-58.771,172.615,22.578,154.091
C02542=1071.028,-72.641,-58.760,172.614,22.576,154.091
C02543=1071.022,-72.891,-58.748,172.612,22.575,154.091
C02544=1071.017,-73.141,-58.738,172.611,22.573,154.090
C02545=1071.010,-73.390,-58.726,172.609,22.571,154.090
C02546=1071.004,-73.640,-58.715,172.608,22.569,154.090
C02547=1070.998,-73.889,-58.704,172.606,22.568,154.090
C02548=1070.992,-74.139,-58.693,172.605,22.566,154.090
C02549=1070.986,-74.389,-58.682,172.603,22.564,154.090
C02550=1070.980,-74.639,-58.671,172.601,22.563,154.090
C02551=1070.974,-74.888,-58.660,172.600,22.561,154.090
C02552=1070.968,-75.137,-58.648,172.598,22.559,154.090
C02553=1070.962,-75.387,-58.637,172.597,22.557,154.090
C02554=1070.956,-75.637,-58.626,172.595,22.556,154.090
C02555=1070.950,-75.887,-58.615,172.594,22.554,154.089
C02556=1070.944,-76.137,-58.604,172.592,22.552,154.089
C02557=1070.938,-76.386,-58.593,172.591,22.551,154.089
C02558=1070.931,-76.636,-58.582,172.589,22.549,154.089
C02559=1070.925,-76.886,-58.571,172.587,22.548,154.089
C02560=1070.919,-77.136,-58.560,172.586,22.546,154.089
C02561=1070.913,-77.385,-58.549,172.584,22.544,154.089
C02562=1070.907,-77.634,-58.538,172.583,22.542,154.089
C02563=1070.901,-77.884,-58.526,172.581,22.541,154.089
C02564=1070.895,-78.134,-58.516,172.580,22.539,154.089
C02565=1070.890,-78.383,-58.505,172.578,22.538,154.089
C02566=1070.883,-78.633,-58.493,172.577,22.536,154.088
C02567=1070.877,-78.883,-58.483,172.575,22.535,154.088
C02568=1070.872,-79.132,-58.472,172.574,22.533,154.088
C02569=1070.865,-79.382,-58.461,172.572,22.531,154.088
C02570=1070.859,-79.632,-58.450,172.571,22.529,154.088
C02571=1070.853,-79.881,-58.439,172.569,22.528,154.088
C02572=1070.847,-80.131,-58.428,172.568,22.526,154.088
C02573=1070.841,-80.381,-58.417,172.566,22.525,154.088
C02574=1070.834,-80.631,-58.407,172.565,22.523,154.088
C02575=1070.828,-80.880,-58.396,172.563,22.521,154.088
C02576=1070.822,-81.130,-58.385,172.562,22.520,154.088
C02577=1070.815,-81.380,-58.374,172.560,22.519,154.088
C02578=1070.810,-81.621,-58.364,172.559,22.517,154.088
C02579=1070.804,-81.862,-58.353,172.557,22.516,154.088
C02580=1070.798,-82.103,-58.343,172.555,22.514,154.088
C02581=1070.792,-82.344,-58.332,172.554,22.512,154.087
C02582=1070.786,-82.585,-58.322,172.552,22.511,154.087
C02583=1070.780,-82.826,-58.311,172.551,22.510,154.087
C02584=1070.774,-83.068,-58.302,172.549,22.508,154.087
C02585=1070.769,-83.309,-58.291,172.548,22.506,154.087
C02586=1070.763,-83.559,-58.280,172.546,22.505,154.087
C02587=1070.756,-83.809,-58.270,172.545,22.504,154.087
C02588=1070.750,-84.058,-58.259,172.543,22.502,154.087
C02589=1070.744,-84.308,-58.248,172.542,22.500,154.087
C02590=1070.737,-84.558,-58.237,172.540,22.499,154.087
C02591=1070.731,-84.807,-58.226,172.539,22.497,154.087
C02592=1070.726,-85.057,-58.215,172.537,22.496,154.087
C02593=1070.719,-85.307,-58.205,172.535,22.494,154.087
C02594=1070.712,-85.604,-58.193,172.533,22.492,154.087
C02595=1070.705,-85.900,-58.180,172.531,22.491,154.087
C02596=1070.697,-86.198,-58.167,172.529,22.488,154.087
C02597=1070.690,-86.495,-58.155,172.527,22.487,154.087
C02598=1070.685,-86.744,-58.144,172.526,22.486,154.087
C02599=1070.677,-86.994,-58.133,172.524,22.484,154.086
C02600=1070.672,-87.243,-58.122,172.523,22.482,154.086
C02601=1070.666,-87.493,-58.113,172.521,22.481,154.086
C02602=1070.660,-87.743,-58.102,172.520,22.480,154.086
C02603=1070.653,-87.993,-58.091,172.518,22.478,154.086
C02604=1070.647,-88.242,-58.080,172.517,22.476,154.086
C02605=1070.642,-88.492,-58.070,172.515,22.475,154.086
C02606=1070.636,-88.742,-58.059,172.513,22.474,154.086
C02607=1070.629,-88.992,-58.049,172.512,22.472,154.086
C02608=1070.623,-89.241,-58.038,172.510,22.470,154.086
C02609=1070.617,-89.491,-58.028,172.509,22.469,154.086
C02610=1070.611,-89.740,-58.017,172.507,22.468,154.086
C02611=1070.605,-89.991,-58.006,172.506,22.466,154.086
C02612=1070.599,-90.240,-57.996,172.504,22.465,154.086
C02613=1070.593,-90.490,-57.986,172.503,22.463,154.086
C02614=1070.586,-90.739,-57.975,172.501,22.462,154.086
C02615=1070.581,-90.989,-57.964,172.499,22.460,154.086
C02616=1070.575,-91.239,-57.954,172.498,22.459,154.086
C02617=1070.568,-91.489,-57.944,172.496,22.458,154.086
C02618=1070.562,-91.738,-57.933,172.495,22.456,154.086
C02619=1070.556,-91.988,-57.923,172.493,22.455,154.086
C02620=1070.550,-92.237,-57.912,172.492,22.453,154.086
C02621=1070.544,-92.487,-57.901,172.490,22.452,154.086
C02622=1070.538,-92.737,-57.892,172.488,22.450,154.085
C02623=1070.532,-92.987,-57.881,172.487,22.449,154.085
C02624=1070.526,-93.237,-57.871,172.485,22.448,154.085
C02625=1070.520,-93.486,-57.860,172.484,22.446,154.085
C02626=1070.514,-93.735,-57.850,172.482,22.445,154.085
C02627=1070.508,-93.986,-57.839,172.480,22.444,154.085
C02628=1070.502,-94.236,-57.829,172.479,22.442,154.085
C02629=1070.496,-94.485,-57.819,172.477,22.440,154.085
C02630=1070.490,-94.735,-57.808,172.476,22.439,154.085
C02631=1070.484,-94.984,-57.798,172.474,22.438,154.085
C02632=1070.478,-95.234,-57.788,172.472,22.436,154.085
C02633=1070.472,-95.483,-57.777,172.471,22.435,154.085
C02634=1070.466,-95.733,-57.767,172.469,22.434,154.085
C02635=1070.459,-95.983,-57.757,172.468,22.432,154.085
C02636=1070.454,-96.233,-57.746,172.466,22.431,154.085
C02637=1070.447,-96.483,-57.736,172.464,22.429,154.085
C02638=1070.442,-96.733,-57.726,172.463,22.428,154.085
C02639=1070.436,-96.982,-57.715,172.461,22.427,154.085
C02640=1070.430,-97.232,-57.705,172.460,22.425,154.085
C02641=1070.424,-97.481,-57.695,172.458,22.424,154.085
C02642=1070.417,-97.763,-57.684,172.456,22.423,154.085
C02643=1070.409,-98.046,-57.671,172.454,22.421,154.085
C02644=1070.403,-98.328,-57.660,172.452,22.420,154.085
C02645=1070.396,-98.610,-57.649,172.451,22.418,154.085
C02646=1070.390,-98.860,-57.639,172.449,22.417,154.085
C02647=1070.384,-99.110,-57.628,172.448,22.416,154.085
C02648=1070.378,-99.360,-57.618,172.446,22.414,154.085
C02649=1070.371,-99.609,-57.608,172.444,22.413,154.085
C02650=1070.366,-99.859,-57.598,172.443,22.411,154.085
C02651=1070.359,-100.109,-57.588,172.441,22.410,154.085
C02652=1070.353,-100.358,-57.578,172.440,22.409,154.085
C02653=1070.347,-100.608,-57.567,172.438,22.407,154.085
C02654=1070.341,-100.858,-57.558,172.436,22.407,154.085
C02655=1070.335,-101.107,-57.548,172.435,22.405,154.085
C02656=1070.328,-101.357,-57.538,172.433,22.404,154.085
C02657=1070.323,-101.607,-57.528,172.431,22.403,154.085
C02658=1070.316,-101.857,-57.517,172.430,22.401,154.085
C02659=1070.310,-102.106,-57.507,172.428,22.400,154.085
C02660=1070.304,-102.357,-57.497,172.426,22.399,154.085
C02661=1070.298,-102.606,-57.487,172.425,22.398,154.085
C02662=1070.292,-102.856,-57.477,172.423,22.396,154.085
C02663=1070.286,-103.106,-57.467,172.422,22.395,154.085
C02664=1070.280,-103.355,-57.457,172.420,22.394,154.085
C02665=1070.274,-103.605,-57.447,172.418,22.393,154.085
C02666=1070.267,-103.854,-57.438,172.417,22.391,154.085
C02667=1070.262,-104.104,-57.427,172.415,22.390,154.085
C02668=1070.256,-104.354,-57.417,172.413,22.389,154.085
C02669=1070.249,-104.603,-57.408,172.412,22.388,154.085
C02670=1070.244,-104.853,-57.397,172.410,22.387,154.085
C02671=1070.237,-105.103,-57.387,172.408,22.385,154.085
C02672=1070.231,-105.353,-57.378,172.407,22.384,154.085
C02673=1070.225,-105.602,-57.368,172.405,22.383,154.085
C02674=1070.219,-105.852,-57.357,172.403,22.382,154.085
C02675=1070.213,-106.102,-57.348,172.403,22.381,154.085
C02676=1070.207,-106.351,-57.338,172.401,22.379,154.085
C02677=1070.201,-106.601,-57.329,172.399,22.379,154.085
C02678=1070.194,-106.851,-57.318,172.398,22.377,154.085
C02679=1070.188,-107.101,-57.308,172.396,22.376,154.085
C02680=1070.182,-107.351,-57.298,172.394,22.375,154.085
C02681=1070.176,-107.601,-57.289,172.393,22.374,154.085
C02682=1070.170,-107.850,-57.278,172.391,22.372,154.085
C02683=1070.163,-108.100,-57.269,172.389,22.372,154.085
C02684=1070.157,-108.350,-57.259,172.388,22.370,154.085
C02685=1070.152,-108.600,-57.249,172.386,22.369,154.085
C02686=1070.146,-108.850,-57.240,172.384,22.368,154.086
C02687=1070.139,-109.099,-57.229,172.383,22.367,154.086
C02688=1070.133,-109.349,-57.220,172.381,22.366,154.086
C02689=1070.127,-109.598,-57.210,172.379,22.365,154.086
C02690=1070.121,-109.848,-57.201,172.378,22.364,154.086
C02691=1070.114,-110.098,-57.191,172.376,22.362,154.086
C02692=1070.108,-110.348,-57.182,172.374,22.361,154.086
C02693=1070.102,-110.597,-57.172,172.373,22.360,154.086
C02694=1070.096,-110.847,-57.162,172.371,22.359,154.086
C02695=1070.090,-111.097,-57.152,172.369,22.358,154.086
C02696=1070.084,-111.347,-57.142,172.368,22.357,154.086
C02697=1070.078,-111.596,-57.132,172.366,22.356,154.086
C02698=1070.072,-111.846,-57.123,172.364,22.355,154.086
C02699=1070.066,-112.095,-57.114,172.362,22.354,154.086
C02700=1070.060,-112.345,-57.104,172.362,22.353,154.086
C02701=1070.054,-112.595,-57.094,172.360,22.352,154.086
C02702=1070.048,-112.845,-57.085,172.358,22.351,154.086
C02703=1070.041,-113.094,-57.075,172.357,22.349,154.086
C02704=1070.035,-113.344,-57.065,172.355,22.349,154.086
C02705=1070.029,-113.593,-57.055,172.353,22.347,154.086
C02706=1070.022,-113.873,-57.045,172.352,22.346,154.086
C02707=1070.015,-114.154,-57.034,172.349,22.345,154.086
C02708=1070.008,-114.434,-57.024,172.347,22.344,154.087
C02709=1070.002,-114.713,-57.013,172.346,22.342,154.086
C02710=1069.996,-114.963,-57.003,172.344,22.342,154.087
C02711=1069.989,-115.213,-56.994,172.342,22.341,154.087
C02712=1069.983,-115.463,-56.984,172.340,22.339,154.087
C02713=1069.977,-115.713,-56.975,172.339,22.339,154.087
C02714=1069.971,-115.962,-56.965,172.337,22.337,154.087
C02715=1069.965,-116.212,-56.955,172.335,22.337,154.087
C02716=1069.959,-116.462,-56.946,172.333,22.336,154.087
C02717=1069.952,-116.712,-56.936,172.333,22.335,154.087
C02718=1069.947,-116.961,-56.927,172.331,22.334,154.087
C02719=1069.941,-117.211,-56.918,172.329,22.333,154.087
C02720=1069.934,-117.461,-56.908,172.328,22.332,154.087
C02721=1069.928,-117.710,-56.898,172.326,22.331,154.087
C02722=1069.922,-117.960,-56.889,172.324,22.330,154.087
C02723=1069.915,-118.210,-56.880,172.322,22.329,154.087
C02724=1069.909,-118.459,-56.870,172.321,22.328,154.088
C02725=1069.903,-118.709,-56.861,172.319,22.327,154.088
C02726=1069.897,-118.959,-56.851,172.317,22.326,154.088
C02727=1069.890,-119.209,-56.842,172.315,22.325,154.088
C02728=1069.885,-119.459,-56.833,172.314,22.324,154.088
C02729=1069.879,-119.708,-56.824,172.312,22.323,154.088
C02730=1069.873,-119.958,-56.814,172.310,22.322,154.088
C02731=1069.867,-120.208,-56.804,172.309,22.321,154.088
C02732=1069.861,-120.458,-56.795,172.308,22.320,154.088
C02733=1069.854,-120.707,-56.786,172.306,22.320,154.088
C02734=1069.847,-120.957,-56.776,172.304,22.319,154.088
C02735=1069.842,-121.206,-56.767,172.302,22.318,154.088
C02736=1069.836,-121.457,-56.758,172.301,22.317,154.088
C02737=1069.830,-121.706,-56.749,172.299,22.316,154.088
C02738=1069.824,-121.956,-56.739,172.297,22.315,154.089
C02739=1069.817,-122.206,-56.730,172.295,22.314,154.089
C02740=1069.811,-122.455,-56.721,172.294,22.313,154.089
C02741=1069.805,-122.706,-56.712,172.292,22.312,154.089
C02742=1069.799,-122.955,-56.703,172.290,22.311,154.089
C02743=1069.793,-123.205,-56.693,172.289,22.311,154.089
C02744=1069.787,-123.455,-56.683,172.287,22.310,154.089
C02745=1069.781,-123.704,-56.674,172.286,22.309,154.089
C02746=1069.774,-123.954,-56.666,172.284,22.308,154.089
C02747=1069.768,-124.203,-56.656,172.282,22.307,154.089
C02748=1069.762,-124.453,-56.647,172.281,22.306,154.089
C02749=1069.756,-124.703,-56.637,172.279,22.306,154.090
C02750=1069.750,-124.954,-56.628,172.277,22.305,154.090
C02751=1069.743,-125.203,-56.619,172.275,22.304,154.090
C02752=1069.737,-125.453,-56.610,172.274,22.303,154.090
C02753=1069.732,-125.702,-56.601,172.272,22.302,154.090
C02754=1069.725,-125.952,-56.592,172.270,22.302,154.090
C02755=1069.719,-126.202,-56.583,172.268,22.300,154.090
C02756=1069.713,-126.452,-56.573,172.267,22.300,154.090
C02757=1069.707,-126.702,-56.564,172.266,22.299,154.090
C02758=1069.700,-126.951,-56.556,172.264,22.298,154.090
C02759=1069.694,-127.201,-56.546,172.262,22.297,154.091
C02760=1069.688,-127.450,-56.537,172.260,22.297,154.091
C02761=1069.682,-127.701,-56.528,172.259,22.296,154.091
C02762=1069.676,-127.951,-56.519,172.257,22.295,154.091
C02763=1069.672,-128.202,-56.509,172.255,22.294,154.091
C02764=1069.669,-128.453,-56.499,172.254,22.291,154.091
C02765=1069.669,-128.703,-56.487,172.253,22.289,154.090
C02766=1069.671,-128.956,-56.474,172.252,22.285,154.090
C02767=1069.674,-129.209,-56.461,172.251,22.280,154.089
C02768=1069.679,-129.460,-56.446,172.252,22.276,154.088
C02769=1069.687,-129.711,-56.432,172.252,22.270,154.087
C02770=1069.297,-129.732,-56.600,172.205,22.411,154.119
C02771=1069.290,-129.482,-56.614,172.205,22.417,154.121
C02772=1069.285,-129.231,-56.629,172.205,22.422,154.121
C02773=1069.281,-128.979,-56.642,172.206,22.427,154.122
C02774=1069.279,-128.725,-56.655,172.207,22.430,154.123
C02775=1069.279,-128.475,-56.666,172.208,22.434,154.123
C02776=1069.281,-128.224,-56.677,172.208,22.435,154.123
C02777=1069.286,-127.973,-56.687,172.210,22.437,154.123
C02778=1069.292,-127.723,-56.696,172.211,22.438,154.123
C02779=1069.298,-127.473,-56.706,172.213,22.439,154.123
C02780=1069.305,-127.224,-56.715,172.215,22.439,154.123
C02781=1069.311,-126.973,-56.724,172.217,22.440,154.123
C02782=1069.317,-126.723,-56.733,172.219,22.441,154.123
C02783=1069.322,-126.474,-56.742,172.220,22.442,154.123
C02784=1069.329,-126.225,-56.751,172.222,22.442,154.123
C02785=1069.335,-125.974,-56.760,172.224,22.443,154.122
C02786=1069.341,-125.724,-56.770,172.226,22.444,154.122
C02787=1069.348,-125.475,-56.779,172.227,22.445,154.122
C02788=1069.353,-125.225,-56.787,172.228,22.445,154.122
C02789=1069.360,-124.976,-56.797,172.230,22.447,154.122
C02790=1069.366,-124.726,-56.806,172.232,22.447,154.122
C02791=1069.373,-124.476,-56.815,172.234,22.448,154.122
C02792=1069.378,-124.226,-56.824,172.235,22.449,154.122
C02793=1069.384,-123.977,-56.833,172.237,22.450,154.122
C02794=1069.390,-123.727,-56.843,172.239,22.451,154.122
C02795=1069.396,-123.477,-56.852,172.241,22.451,154.121
C02796=1069.402,-123.227,-56.861,172.242,22.453,154.121
C02797=1069.409,-122.977,-56.870,172.244,22.453,154.121
C02798=1069.415,-122.727,-56.880,172.246,22.454,154.121
C02799=1069.421,-122.478,-56.889,172.248,22.455,154.121
C02800=1069.427,-122.229,-56.899,172.250,22.456,154.121
C02801=1069.433,-121.979,-56.908,172.250,22.457,154.121
C02802=1069.439,-121.728,-56.917,172.252,22.458,154.121
C02803=1069.446,-121.479,-56.926,172.254,22.458,154.121
C02804=1069.452,-121.229,-56.936,172.256,22.459,154.121
C02805=1069.458,-120.979,-56.945,172.257,22.461,154.121
C02806=1069.464,-120.730,-56.954,172.259,22.461,154.121
C02807=1069.470,-120.480,-56.964,172.261,22.462,154.121
C02808=1069.476,-120.230,-56.973,172.263,22.463,154.120
C02809=1069.482,-119.980,-56.982,172.264,22.464,154.120
C02810=1069.488,-119.730,-56.992,172.266,22.465,154.120
C02811=1069.495,-119.481,-57.001,172.268,22.466,154.120
C02812=1069.501,-119.231,-57.010,172.269,22.467,154.120
C02813=1069.507,-118.982,-57.020,172.271,22.468,154.120
C02814=1069.513,-118.732,-57.029,172.273,22.469,154.120
C02815=1069.519,-118.482,-57.039,172.274,22.470,154.120
C02816=1069.526,-118.233,-57.048,172.275,22.470,154.120
C02817=1069.532,-117.983,-57.058,172.277,22.471,154.120
C02818=1069.538,-117.733,-57.067,172.279,22.473,154.120
C02819=1069.544,-117.483,-57.076,172.281,22.473,154.120
C02820=1069.550,-117.233,-57.086,172.282,22.474,154.120
C02821=1069.556,-116.983,-57.095,172.284,22.476,154.120
C02822=1069.562,-116.733,-57.105,172.286,22.476,154.119
C02823=1069.568,-116.484,-57.114,172.288,22.477,154.119
C02824=1069.574,-116.234,-57.124,172.289,22.478,154.119
C02825=1069.580,-115.984,-57.133,172.291,22.479,154.119
C02826=1069.586,-115.735,-57.143,172.293,22.481,154.119
C02827=1069.592,-115.485,-57.153,172.294,22.481,154.119
C02828=1069.599,-115.235,-57.161,172.296,22.482,154.119
C02829=1069.606,-114.986,-57.171,172.298,22.484,154.119
C02830=1069.612,-114.736,-57.181,172.300,22.484,154.119
C02831=1069.618,-114.456,-57.191,172.301,22.486,154.119
C02832=1069.625,-114.175,-57.202,172.303,22.486,154.119
C02833=1069.632,-113.896,-57.214,172.305,22.488,154.119
C02834=1069.639,-113.616,-57.224,172.306,22.489,154.119
C02835=1069.645,-113.367,-57.233,172.308,22.490,154.119
C02836=1069.651,-113.116,-57.244,172.310,22.491,154.119
C02837=1069.657,-112.867,-57.253,172.311,22.492,154.119
C02838=1069.663,-112.617,-57.263,172.313,22.493,154.119
C02839=1069.669,-112.367,-57.272,172.315,22.494,154.119
C02840=1069.675,-112.117,-57.282,172.317,22.495,154.118
C02841=1069.682,-111.867,-57.291,172.318,22.496,154.118
C02842=1069.688,-111.618,-57.301,172.320,22.497,154.118
C02843=1069.694,-111.368,-57.311,172.322,22.499,154.118
C02844=1069.700,-111.119,-57.321,172.323,22.500,154.118
C02845=1069.707,-110.869,-57.330,172.325,22.501,154.118
C02846=1069.713,-110.619,-57.340,172.327,22.502,154.118
C02847=1069.719,-110.369,-57.350,172.328,22.503,154.118
C02848=1069.724,-110.119,-57.360,172.330,22.504,154.118
C02849=1069.730,-109.869,-57.369,172.332,22.505,154.118
C02850=1069.737,-109.620,-57.379,172.333,22.506,154.118
C02851=1069.743,-109.370,-57.389,172.335,22.508,154.118
C02852=1069.749,-109.121,-57.399,172.337,22.508,154.118
C02853=1069.755,-108.871,-57.408,172.338,22.510,154.118
C02854=1069.762,-108.621,-57.418,172.340,22.511,154.118
C02855=1069.768,-108.371,-57.427,172.342,22.512,154.118
C02856=1069.774,-108.121,-57.437,172.342,22.513,154.118
C02857=1069.780,-107.872,-57.448,172.344,22.514,154.118
C02858=1069.786,-107.622,-57.457,172.346,22.515,154.118
C02859=1069.792,-107.372,-57.467,172.347,22.516,154.118
C02860=1069.798,-107.123,-57.477,172.349,22.517,154.118
C02861=1069.805,-106.873,-57.487,172.351,22.518,154.118
C02862=1069.810,-106.623,-57.497,172.352,22.520,154.118
C02863=1069.816,-106.373,-57.507,172.354,22.521,154.118
C02864=1069.822,-106.124,-57.516,172.356,22.522,154.118
C02865=1069.829,-105.874,-57.526,172.357,22.523,154.118
C02866=1069.835,-105.625,-57.536,172.359,22.525,154.118
C02867=1069.841,-105.375,-57.546,172.361,22.525,154.118
C02868=1069.847,-105.125,-57.556,172.362,22.527,154.118
C02869=1069.853,-104.876,-57.566,172.364,22.528,154.118
C02870=1069.859,-104.626,-57.576,172.366,22.530,154.118
C02871=1069.865,-104.376,-57.586,172.367,22.530,154.118
C02872=1069.871,-104.127,-57.596,172.369,22.532,154.118
C02873=1069.877,-103.877,-57.606,172.371,22.533,154.118
C02874=1069.884,-103.626,-57.616,172.372,22.534,154.118
C02875=1069.890,-103.377,-57.626,172.374,22.535,154.117
C02876=1069.896,-103.127,-57.636,172.376,22.536,154.117
C02877=1069.902,-102.877,-57.646,172.377,22.538,154.118
C02878=1069.908,-102.628,-57.656,172.379,22.539,154.118
C02879=1069.914,-102.378,-57.666,172.381,22.541,154.118
C02880=1069.920,-102.128,-57.676,172.382,22.542,154.118
C02881=1069.926,-101.879,-57.686,172.384,22.543,154.117
C02882=1069.932,-101.629,-57.696,172.386,22.544,154.117
C02883=1069.939,-101.380,-57.706,172.387,22.545,154.117
C02884=1069.944,-101.129,-57.716,172.389,22.547,154.117
C02885=1069.950,-100.880,-57.726,172.390,22.548,154.117
C02886=1069.957,-100.630,-57.736,172.392,22.549,154.118
C02887=1069.963,-100.380,-57.747,172.394,22.550,154.117
C02888=1069.969,-100.130,-57.757,172.395,22.552,154.117
C02889=1069.976,-99.881,-57.767,172.397,22.553,154.117
C02890=1069.982,-99.631,-57.776,172.399,22.554,154.117
C02891=1069.987,-99.381,-57.787,172.400,22.556,154.117
C02892=1069.994,-99.132,-57.797,172.402,22.557,154.117
C02893=1069.999,-98.882,-57.808,172.403,22.558,154.117
C02894=1070.006,-98.632,-57.817,172.405,22.560,154.118
C02895=1070.013,-98.349,-57.829,172.407,22.561,154.118
C02896=1070.020,-98.068,-57.841,172.408,22.562,154.118
C02897=1070.027,-97.786,-57.852,172.410,22.564,154.118
C02898=1070.034,-97.503,-57.863,172.412,22.565,154.118
C02899=1070.040,-97.253,-57.874,172.414,22.567,154.118
C02900=1070.046,-97.003,-57.884,172.416,22.568,154.118
C02901=1070.052,-96.754,-57.895,172.417,22.569,154.118
C02902=1070.058,-96.504,-57.904,172.419,22.571,154.118
C02903=1070.064,-96.255,-57.915,172.420,22.572,154.118
C02904=1070.070,-96.005,-57.925,172.422,22.574,154.118
C02905=1070.076,-95.755,-57.935,172.424,22.575,154.118
C02906=1070.082,-95.505,-57.946,172.425,22.576,154.118
C02907=1070.088,-95.255,-57.956,172.427,22.578,154.118
C02908=1070.094,-95.006,-57.967,172.428,22.579,154.118
C02909=1070.100,-94.756,-57.977,172.430,22.581,154.118
C02910=1070.106,-94.507,-57.988,172.431,22.582,154.118
C02911=1070.112,-94.257,-57.997,172.433,22.584,154.118
C02912=1070.118,-94.007,-58.008,172.435,22.585,154.118
C02913=1070.125,-93.757,-58.019,172.436,22.586,154.118
C02914=1070.130,-93.507,-58.029,172.438,22.588,154.118
C02915=1070.136,-93.258,-58.040,172.440,22.589,154.118
C02916=1070.142,-93.008,-58.049,172.441,22.590,154.118
C02917=1070.148,-92.759,-58.060,172.443,22.592,154.118
C02918=1070.154,-92.509,-58.070,172.444,22.594,154.118
C02919=1070.160,-92.259,-58.081,172.446,22.595,154.118
C02920=1070.167,-92.009,-58.091,172.447,22.596,154.118
C02921=1070.173,-91.760,-58.102,172.449,22.598,154.118
C02922=1070.178,-91.510,-58.112,172.451,22.599,154.118
C02923=1070.184,-91.261,-58.123,172.452,22.600,154.118
C02924=1070.191,-91.010,-58.134,172.454,22.602,154.118
C02925=1070.197,-90.761,-58.143,172.455,22.604,154.118
C02926=1070.203,-90.511,-58.154,172.457,22.605,154.118
C02927=1070.208,-90.262,-58.165,172.458,22.606,154.118
C02928=1070.215,-90.012,-58.175,172.460,22.608,154.118
C02929=1070.221,-89.762,-58.186,172.461,22.609,154.119
C02930=1070.227,-89.512,-58.196,172.463,22.611,154.119
C02931=1070.233,-89.263,-58.207,172.465,22.612,154.119
C02932=1070.239,-89.013,-58.217,172.466,22.614,154.119
C02933=1070.246,-88.763,-58.228,172.468,22.615,154.119
C02934=1070.251,-88.514,-58.239,172.469,22.617,154.119
C02935=1070.257,-88.264,-58.250,172.471,22.618,154.119
C02936=1070.263,-88.014,-58.259,172.473,22.619,154.119
C02937=1070.270,-87.764,-58.271,172.474,22.621,154.119
C02938=1070.276,-87.515,-58.281,172.476,22.622,154.119
C02939=1070.282,-87.265,-58.292,172.477,22.624,154.119
C02940=1070.288,-87.016,-58.303,172.479,22.625,154.119
C02941=1070.294,-86.765,-58.312,172.480,22.627,154.119
C02942=1070.300,-86.516,-58.323,172.482,22.628,154.119
C02943=1070.306,-86.266,-58.334,172.483,22.630,154.119
C02944=1070.313,-86.017,-58.345,172.485,22.631,154.119
C02945=1070.319,-85.767,-58.356,172.487,22.633,154.119
C02946=1070.324,-85.517,-58.366,172.488,22.635,154.119
C02947=1070.331,-85.268,-58.376,172.490,22.636,154.119
C02948=1070.337,-85.018,-58.387,172.491,22.637,154.119
C02949=1070.343,-84.768,-58.398,172.493,22.639,154.119
C02950=1070.349,-84.519,-58.409,172.494,22.641,154.120
C02951=1070.356,-84.269,-58.420,172.496,22.642,154.120
C02952=1070.361,-84.019,-58.431,172.498,22.643,154.120
C02953=1070.368,-83.770,-58.441,172.499,22.645,154.120
C02954=1070.374,-83.519,-58.452,172.501,22.646,154.120
C02955=1070.380,-83.270,-58.462,172.502,22.648,154.120
C02956=1070.386,-83.021,-58.473,172.504,22.650,154.120
C02957=1070.392,-82.770,-58.484,172.505,22.651,154.120
C02958=1070.398,-82.521,-58.495,172.507,22.652,154.120
C02959=1070.405,-82.241,-58.507,172.509,22.655,154.120
C02960=1070.412,-81.961,-58.519,172.511,22.656,154.120
C02961=1070.419,-81.681,-58.531,172.512,22.658,154.120
C02962=1070.426,-81.400,-58.543,172.514,22.659,154.120
C02963=1070.432,-81.151,-58.553,172.515,22.661,154.120
C02964=1070.438,-80.902,-58.564,172.518,22.663,154.120
C02965=1070.444,-80.651,-58.576,172.519,22.664,154.120
C02966=1070.451,-80.402,-58.586,172.521,22.666,154.120
C02967=1070.457,-80.152,-58.597,172.522,22.668,154.120
C02968=1070.463,-79.903,-58.608,172.524,22.669,154.121
C02969=1070.469,-79.653,-58.619,172.525,22.671,154.121
C02970=1070.475,-79.403,-58.630,172.527,22.673,154.121
C02971=1070.481,-79.153,-58.641,172.529,22.674,154.121
C02972=1070.487,-78.904,-58.651,172.530,22.676,154.121
C02973=1070.494,-78.654,-58.663,172.532,22.677,154.121
C02974=1070.499,-78.405,-58.673,172.533,22.679,154.121
C02975=1070.505,-78.155,-58.684,172.535,22.681,154.121
C02976=1070.511,-77.905,-58.696,172.536,22.682,154.121
C02977=1070.518,-77.656,-58.707,172.538,22.684,154.121
C02978=1070.524,-77.406,-58.718,172.539,22.686,154.121
C02979=1070.530,-77.156,-58.729,172.541,22.687,154.121
C02980=1070.535,-76.907,-58.740,172.542,22.689,154.122
C02981=1070.542,-76.657,-58.751,172.544,22.690,154.122
C02982=1070.548,-76.407,-58.762,172.545,22.692,154.122
C02983=1070.554,-76.158,-58.773,172.547,22.694,154.122
C02984=1070.560,-75.908,-58.784,172.548,22.695,154.122
C02985=1070.566,-75.658,-58.795,172.550,22.697,154.122
C02986=1070.572,-75.408,-58.806,172.551,22.699,154.122
C02987=1070.578,-75.159,-58.817,172.553,22.701,154.122
C02988=1070.585,-74.909,-58.829,172.554,22.702,154.122
C02989=1070.590,-74.660,-58.840,172.556,22.704,154.122
C02990=1070.596,-74.410,-58.850,172.557,22.706,154.123
C02991=1070.603,-74.160,-58.862,172.559,22.707,154.123
C02992=1070.608,-73.910,-58.873,172.561,22.709,154.123
C02993=1070.615,-73.661,-58.885,172.563,22.711,154.123
C02994=1070.621,-73.411,-58.895,172.564,22.713,154.123
C02995=1070.626,-73.162,-58.906,172.566,22.715,154.123
C02996=1070.633,-72.912,-58.918,172.567,22.716,154.123
C02997=1070.638,-72.662,-58.929,172.569,22.718,154.123
C02998=1070.644,-72.412,-58.941,172.570,22.720,154.123
C02999=1070.650,-72.163,-58.952,172.571,22.722,154.123
C03000=1070.656,-71.913,-58.963,172.573,22.723,154.124
C03001=1070.662,-71.663,-58.974,172.575,22.725,154.124
C03002=1070.668,-71.414,-58.985,172.576,22.727,154.124
C03003=1070.675,-71.164,-58.997,172.577,22.729,154.124
C03004=1070.680,-70.914,-59.008,172.579,22.731,154.124
C03005=1070.685,-70.665,-59.019,172.580,22.732,154.124
C03006=1070.692,-70.415,-59.031,172.582,22.734,154.124
C03007=1070.698,-70.166,-59.042,172.583,22.736,154.124
C03008=1070.704,-69.915,-59.053,172.585,22.738,154.125
C03009=1070.710,-69.666,-59.064,172.586,22.739,154.125
C03010=1070.716,-69.416,-59.077,172.588,22.741,154.125
C03011=1070.721,-69.167,-59.088,172.589,22.743,154.125
C03012=1070.727,-68.917,-59.098,172.591,22.745,154.125
C03013=1070.734,-68.668,-59.110,172.593,22.747,154.125
C03014=1070.740,-68.418,-59.121,172.594,22.749,154.125
C03015=1070.745,-68.168,-59.133,172.596,22.750,154.125
C03016=1070.751,-67.919,-59.145,172.597,22.752,154.125
C03017=1070.758,-67.668,-59.156,172.599,22.754,154.126
C03018=1070.763,-67.419,-59.167,172.600,22.756,154.126
C03019=1070.770,-67.169,-59.179,172.602,22.758,154.126
C03020=1070.775,-66.920,-59.190,172.603,22.760,154.126
C03021=1070.782,-66.670,-59.202,172.605,22.761,154.126
C03022=1070.787,-66.421,-59.213,172.606,22.763,154.126
C03023=1070.795,-66.143,-59.226,172.608,22.765,154.126
C03024=1070.801,-65.865,-59.239,172.610,22.767,154.126
C03025=1070.807,-65.587,-59.251,172.611,22.769,154.127
C03026=1070.814,-65.309,-59.264,172.613,22.771,154.127
C03027=1070.820,-65.060,-59.276,172.614,22.773,154.127
C03028=1070.826,-64.810,-59.287,172.616,22.775,154.127
C03029=1070.833,-64.560,-59.299,172.617,22.777,154.127
C03030=1070.838,-64.310,-59.311,172.619,22.778,154.127
C03031=1070.844,-64.061,-59.322,172.620,22.780,154.127
C03032=1070.850,-63.811,-59.333,172.622,22.783,154.128
C03033=1070.857,-63.562,-59.345,172.624,22.785,154.128
C03034=1070.863,-63.312,-59.356,172.625,22.786,154.128
C03035=1070.868,-63.062,-59.369,172.627,22.788,154.128
C03036=1070.874,-62.813,-59.380,172.628,22.790,154.128
C03037=1070.881,-62.563,-59.392,172.630,22.792,154.128
C03038=1070.887,-62.314,-59.402,172.631,22.793,154.128
C03039=1070.892,-62.064,-59.415,172.633,22.795,154.128
C03040=1070.899,-61.814,-59.426,172.634,22.797,154.129
C03041=1070.905,-61.565,-59.438,172.635,22.799,154.129
C03042=1070.910,-61.314,-59.450,172.637,22.801,154.129
C03043=1070.917,-61.065,-59.461,172.638,22.803,154.129
C03044=1070.923,-60.815,-59.473,172.640,22.805,154.129
C03045=1070.929,-60.566,-59.484,172.641,22.807,154.129
C03046=1070.934,-60.316,-59.496,172.643,22.809,154.130
C03047=1070.941,-60.066,-59.508,172.644,22.811,154.130
C03048=1070.947,-59.817,-59.519,172.647,22.812,154.130
C03049=1070.953,-59.567,-59.531,172.648,22.814,154.130
C03050=1070.959,-59.317,-59.543,172.649,22.816,154.130
C03051=1070.965,-59.068,-59.554,172.651,22.818,154.130
C03052=1070.972,-58.818,-59.566,172.652,22.820,154.130
C03053=1070.978,-58.568,-59.579,172.654,22.822,154.130
C03054=1070.983,-58.319,-59.590,172.655,22.824,154.131
C03055=1070.990,-58.069,-59.602,172.657,22.826,154.131
C03056=1070.996,-57.819,-59.613,172.658,22.827,154.131
C03057=1071.002,-57.570,-59.625,172.660,22.829,154.131
C03058=1071.008,-57.320,-59.637,172.661,22.831,154.131
C03059=1071.014,-57.070,-59.649,172.662,22.833,154.131
C03060=1071.020,-56.821,-59.660,172.664,22.835,154.131
C03061=1071.027,-56.571,-59.672,172.665,22.837,154.132
C03062=1071.032,-56.321,-59.684,172.667,22.839,154.132
C03063=1071.038,-56.072,-59.696,172.669,22.841,154.132
C03064=1071.045,-55.822,-59.708,172.671,22.843,154.132
C03065=1071.051,-55.572,-59.720,172.672,22.845,154.132
C03066=1071.057,-55.323,-59.731,172.673,22.847,154.132
C03067=1071.063,-55.073,-59.743,172.675,22.849,154.132
C03068=1071.069,-54.824,-59.756,172.676,22.851,154.133
C03069=1071.075,-54.574,-59.767,172.678,22.852,154.133
C03070=1071.082,-54.324,-59.778,172.679,22.854,154.133
C03071=1071.087,-54.075,-59.791,172.681,22.856,154.133
C03072=1071.094,-53.825,-59.803,172.682,22.858,154.133
C03073=1071.100,-53.576,-59.814,172.683,22.860,154.133
C03074=1071.106,-53.326,-59.826,172.685,22.862,154.133
C03075=1071.112,-53.076,-59.838,172.686,22.864,154.134
C03076=1071.119,-52.827,-59.850,172.688,22.866,154.134
C03077=1071.124,-52.577,-59.863,172.690,22.869,154.134
C03078=1071.131,-52.327,-59.874,172.691,22.870,154.134
C03079=1071.137,-52.078,-59.886,172.693,22.872,154.134
C03080=1071.143,-51.828,-59.898,172.694,22.874,154.134
C03081=1071.149,-51.579,-59.910,172.696,22.876,154.135
C03082=1071.155,-51.329,-59.922,172.697,22.878,154.135
C03083=1071.162,-51.097,-59.933,172.699,22.880,154.135
C03084=1071.167,-50.864,-59.945,172.700,22.882,154.135
C03085=1071.172,-50.633,-59.956,172.701,22.884,154.135
C03086=1071.179,-50.400,-59.966,172.703,22.886,154.135
C03087=1071.184,-50.168,-59.978,172.704,22.887,154.135
C03088=1071.190,-49.937,-59.989,172.705,22.889,154.136
C03089=1071.195,-49.704,-60.001,172.706,22.891,154.136
C03090=1071.204,-49.348,-60.018,172.708,22.894,154.136
C03091=1071.213,-48.974,-60.037,172.711,22.897,154.136
C03092=1071.219,-48.724,-60.048,172.713,22.899,154.136
C03093=1071.224,-48.475,-60.060,172.714,22.901,154.137
C03094=1071.230,-48.225,-60.073,172.716,22.903,154.137
C03095=1071.237,-47.976,-60.085,172.717,22.905,154.137
C03096=1071.242,-47.726,-60.097,172.718,22.908,154.137
C03097=1071.248,-47.477,-60.109,172.720,22.909,154.137
C03098=1071.255,-47.227,-60.121,172.721,22.911,154.138
C03099=1071.261,-46.977,-60.134,172.723,22.914,154.138
C03100=1071.266,-46.728,-60.146,172.724,22.916,154.138
C03101=1071.272,-46.478,-60.158,172.725,22.918,154.138
C03102=1071.278,-46.228,-60.171,172.727,22.919,154.138
C03103=1071.284,-45.979,-60.183,172.728,22.922,154.139
C03104=1071.291,-45.729,-60.195,172.730,22.924,154.139
C03105=1071.296,-45.480,-60.207,172.732,22.926,154.139
C03106=1071.302,-45.230,-60.220,172.733,22.928,154.139
C03107=1071.309,-44.980,-60.232,172.735,22.930,154.139
C03108=1071.315,-44.731,-60.244,172.736,22.932,154.139
C03109=1071.320,-44.481,-60.257,172.737,22.935,154.140
C03110=1071.327,-44.232,-60.268,172.739,22.937,154.140
C03111=1071.333,-43.982,-60.281,172.740,22.938,154.140
C03112=1071.338,-43.732,-60.294,172.742,22.940,154.140
C03113=1071.344,-43.482,-60.306,172.743,22.943,154.140
C03114=1071.350,-43.233,-60.318,172.744,22.945,154.141
C03115=1071.356,-42.983,-60.330,172.746,22.947,154.141
C03116=1071.363,-42.734,-60.344,172.747,22.949,154.141
C03117=1071.369,-42.485,-60.356,172.749,22.951,154.141
C03118=1071.375,-42.235,-60.368,172.751,22.953,154.141
C03119=1071.381,-41.985,-60.381,172.752,22.956,154.141
C03120=1071.386,-41.736,-60.393,172.754,22.958,154.142
C03121=1071.393,-41.486,-60.405,172.755,22.959,154.142
C03122=1071.399,-41.236,-60.417,172.756,22.962,154.142
C03123=1071.405,-40.986,-60.430,172.758,22.964,154.142
C03124=1071.411,-40.737,-60.443,172.759,22.966,154.142
C03125=1071.418,-40.487,-60.455,172.760,22.968,154.143
C03126=1071.424,-40.238,-60.468,172.762,22.970,154.143
C03127=1071.429,-39.988,-60.480,172.763,22.972,154.143
C03128=1071.435,-39.738,-60.492,172.765,22.974,154.143
C03129=1071.441,-39.489,-60.504,172.767,22.977,154.143
C03130=1071.448,-39.240,-60.518,172.768,22.979,154.144
C03131=1071.454,-38.990,-60.530,172.770,22.981,154.144
C03132=1071.459,-38.740,-60.543,172.771,22.983,154.144
C03133=1071.466,-38.490,-60.555,172.772,22.985,154.144
C03134=1071.472,-38.240,-60.567,172.774,22.987,154.144
C03135=1071.478,-37.991,-60.581,172.775,22.990,154.145
C03136=1071.484,-37.742,-60.593,172.777,22.991,154.145
C03137=1071.489,-37.492,-60.605,172.778,22.994,154.145
C03138=1071.495,-37.242,-60.618,172.779,22.996,154.145
C03139=1071.502,-36.993,-60.631,172.780,22.998,154.145
C03140=1071.507,-36.743,-60.644,172.783,23.000,154.146
C03141=1071.513,-36.493,-60.656,172.784,23.003,154.146
C03142=1071.519,-36.243,-60.669,172.786,23.005,154.146
C03143=1071.525,-35.994,-60.682,172.787,23.007,154.146
C03144=1071.531,-35.745,-60.694,172.788,23.009,154.146
C03145=1071.537,-35.495,-60.707,172.790,23.012,154.147
C03146=1071.543,-35.246,-60.720,172.791,23.013,154.147
C03147=1071.549,-34.996,-60.733,172.792,23.016,154.147
C03148=1071.555,-34.746,-60.745,172.794,23.018,154.147
C03149=1071.561,-34.497,-60.758,172.795,23.020,154.148
C03150=1071.567,-34.247,-60.771,172.796,23.022,154.148
C03151=1071.574,-33.971,-60.785,172.799,23.025,154.148
C03152=1071.580,-33.695,-60.799,172.800,23.027,154.148
C03153=1071.587,-33.419,-60.814,172.801,23.030,154.149
C03154=1071.594,-33.143,-60.827,172.803,23.033,154.149
C03155=1071.600,-32.893,-60.840,172.805,23.035,154.149
C03156=1071.606,-32.643,-60.853,172.806,23.037,154.149
C03157=1071.612,-32.394,-60.865,172.807,23.039,154.149
C03158=1071.618,-32.144,-60.878,172.809,23.041,154.150
C03159=1071.624,-31.895,-60.891,172.810,23.043,154.150
C03160=1071.630,-31.645,-60.904,172.811,23.046,154.150
C03161=1071.636,-31.395,-60.916,172.813,23.048,154.150
C03162=1071.642,-31.146,-60.930,172.814,23.050,154.150
C03163=1071.647,-30.896,-60.943,172.815,23.052,154.151
C03164=1071.653,-30.647,-60.956,172.818,23.055,154.151
C03165=1071.659,-30.397,-60.969,172.819,23.057,154.151
C03166=1071.665,-30.147,-60.982,172.821,23.059,154.151
C03167=1071.671,-29.898,-60.994,172.822,23.061,154.152
C03168=1071.677,-29.648,-61.008,172.823,23.063,154.152
C03169=1071.683,-29.398,-61.020,172.825,23.066,154.152
C03170=1071.690,-29.149,-61.034,172.826,23.068,154.152
C03171=1071.695,-28.899,-61.046,172.827,23.070,154.152
C03172=1071.702,-28.650,-61.059,172.829,23.072,154.153
C03173=1071.708,-28.400,-61.072,172.830,23.074,154.153
C03174=1071.714,-28.151,-61.085,172.831,23.077,154.153
C03175=1071.720,-27.901,-61.098,172.834,23.079,154.153
C03176=1071.726,-27.652,-61.111,172.835,23.082,154.154
C03177=1071.732,-27.402,-61.124,172.836,23.084,154.154
C03178=1071.739,-27.152,-61.137,172.838,23.086,154.154
C03179=1071.745,-26.902,-61.150,172.839,23.088,154.154
C03180=1071.751,-26.653,-61.163,172.840,23.090,154.154
C03181=1071.757,-26.403,-61.176,172.842,23.093,154.155
C03182=1071.762,-26.153,-61.189,172.843,23.095,154.155
C03183=1071.768,-25.904,-61.203,172.844,23.097,154.155
C03184=1071.774,-25.654,-61.215,172.846,23.099,154.155
C03185=1071.780,-25.405,-61.229,172.847,23.102,154.156
C03186=1071.786,-25.155,-61.242,172.849,23.105,154.156
C03187=1071.792,-24.905,-61.255,172.851,23.106,154.156
C03188=1071.798,-24.656,-61.268,172.852,23.109,154.156
C03189=1071.804,-24.406,-61.281,172.853,23.111,154.157
C03190=1071.809,-24.157,-61.295,172.855,23.113,154.157
C03191=1071.816,-23.907,-61.308,172.856,23.116,154.157
C03192=1071.822,-23.658,-61.320,172.857,23.118,154.157
C03193=1071.828,-23.408,-61.334,172.858,23.121,154.158
C03194=1071.833,-23.159,-61.348,172.860,23.122,154.158
C03195=1071.839,-22.909,-61.360,172.861,23.125,154.158
C03196=1071.845,-22.660,-61.373,172.863,23.128,154.158
C03197=1071.851,-22.410,-61.387,172.865,23.130,154.159
C03198=1071.857,-22.160,-61.400,172.866,23.132,154.159
C03199=1071.863,-21.911,-61.413,172.867,23.134,154.159
C03200=1071.869,-21.662,-61.426,172.869,23.137,154.159
C03201=1071.875,-21.412,-61.440,172.870,23.139,154.159
C03202=1071.881,-21.162,-61.453,172.871,23.141,154.160
C03203=1071.887,-20.912,-61.466,172.873,23.144,154.160
C03204=1071.893,-20.663,-61.480,172.874,23.146,154.160
C03205=1071.899,-20.413,-61.494,172.875,23.148,154.160
C03206=1071.905,-20.163,-61.506,172.877,23.150,154.161
C03207=1071.911,-19.914,-61.519,172.879,23.153,154.161
C03208=1071.917,-19.665,-61.533,172.880,23.156,154.161
C03209=1071.923,-19.415,-61.547,172.882,23.157,154.161
C03210=1071.929,-19.166,-61.560,172.883,23.160,154.162
C03211=1071.934,-18.916,-61.573,172.884,23.162,154.162
C03212=1071.941,-18.666,-61.587,172.885,23.165,154.162
C03213=1071.947,-18.417,-61.600,172.887,23.167,154.162
C03214=1071.953,-18.167,-61.614,172.888,23.169,154.163
C03215=1071.959,-17.891,-61.628,172.890,23.172,154.163
C03216=1071.967,-17.614,-61.643,172.892,23.174,154.163
C03217=1071.973,-17.336,-61.659,172.893,23.177,154.163
C03218=1071.980,-17.060,-61.673,172.895,23.180,154.164
C03219=1071.986,-16.810,-61.686,172.896,23.182,154.164
C03220=1071.992,-16.560,-61.700,172.898,23.184,154.164
C03221=1071.998,-16.310,-61.713,172.899,23.187,154.165
C03222=1072.004,-16.061,-61.726,172.900,23.189,154.165
C03223=1072.010,-15.812,-61.740,172.902,23.191,154.165
C03224=1072.016,-15.562,-61.754,172.903,23.194,154.165
C03225=1072.022,-15.313,-61.767,172.904,23.196,154.166
C03226=1072.028,-15.063,-61.781,172.905,23.198,154.166
C03227=1072.034,-14.814,-61.794,172.907,23.200,154.166
C03228=1072.040,-14.564,-61.808,172.909,23.203,154.166
C03229=1072.046,-14.314,-61.821,172.910,23.206,154.166
C03230=1072.051,-14.064,-61.835,172.912,23.208,154.167
C03231=1072.057,-13.815,-61.848,172.913,23.210,154.167
C03232=1072.064,-13.565,-61.862,172.914,23.213,154.167
C03233=1072.069,-13.315,-61.876,172.916,23.215,154.168
C03234=1072.075,-13.066,-61.889,172.917,23.218,154.168
C03235=1072.081,-12.817,-61.903,172.918,23.220,154.168
C03236=1072.087,-12.567,-61.916,172.920,23.222,154.168
C03237=1072.092,-12.318,-61.930,172.921,23.224,154.169
C03238=1072.099,-12.068,-61.944,172.923,23.227,154.169
C03239=1072.105,-11.818,-61.958,172.924,23.230,154.169
C03240=1072.111,-11.569,-61.971,172.926,23.232,154.169
C03241=1072.116,-11.319,-61.985,172.927,23.234,154.170
C03242=1072.123,-11.070,-61.998,172.928,23.237,154.170
C03243=1072.129,-10.820,-62.012,172.929,23.239,154.170
C03244=1072.134,-10.571,-62.027,172.931,23.242,154.171
C03245=1072.141,-10.322,-62.040,172.932,23.244,154.171
C03246=1072.146,-10.072,-62.054,172.934,23.246,154.171
C03247=1072.153,-9.822,-62.068,172.935,23.248,154.171
C03248=1072.158,-9.572,-62.082,172.937,23.251,154.171
C03249=1072.165,-9.323,-62.095,172.938,23.254,154.172
C03250=1072.170,-9.074,-62.109,172.940,23.256,154.172
C03251=1072.176,-8.823,-62.123,172.941,23.259,154.172
C03252=1072.182,-8.574,-62.136,172.942,23.261,154.173
C03253=1072.188,-8.324,-62.150,172.943,23.263,154.173
C03254=1072.194,-8.076,-62.164,172.945,23.266,154.173
C03255=1072.200,-7.826,-62.178,172.946,23.268,154.173
C03256=1072.206,-7.576,-62.192,172.947,23.270,154.174
C03257=1072.212,-7.327,-62.205,172.949,23.273,154.174
C03258=1072.218,-7.077,-62.219,172.951,23.275,154.174
C03259=1072.224,-6.827,-62.233,172.952,23.278,154.174
C03260=1072.230,-6.578,-62.248,172.954,23.280,154.175
C03261=1072.236,-6.329,-62.261,172.955,23.283,154.175
C03262=1072.243,-6.079,-62.275,172.956,23.285,154.175
C03263=1072.248,-5.829,-62.289,172.957,23.287,154.176
C03264=1072.253,-5.580,-62.303,172.959,23.290,154.176
C03265=1072.260,-5.331,-62.317,172.960,23.292,154.176
C03266=1072.266,-5.081,-62.331,172.961,23.295,154.176
C03267=1072.272,-4.831,-62.344,172.963,23.297,154.177
C03268=1072.278,-4.582,-62.358,172.965,23.299,154.177
C03269=1072.284,-4.331,-62.372,172.966,23.302,154.177
C03270=1072.290,-4.083,-62.386,172.968,23.304,154.177
C03271=1072.296,-3.833,-62.400,172.969,23.307,154.178
C03272=1072.302,-3.583,-62.414,172.970,23.309,154.178
C03273=1072.308,-3.334,-62.428,172.971,23.312,154.178
C03274=1072.314,-3.085,-62.442,172.973,23.314,154.178
C03275=1072.320,-2.834,-62.457,172.974,23.316,154.179
C03276=1072.325,-2.585,-62.470,172.975,23.319,154.179
C03277=1072.331,-2.336,-62.485,172.977,23.322,154.179
C03278=1072.337,-2.086,-62.499,172.979,23.324,154.180
C03279=1072.344,-1.808,-62.515,172.980,23.327,154.180
C03280=1072.350,-1.529,-62.530,172.981,23.329,154.180
C03281=1072.357,-1.251,-62.546,172.983,23.333,154.181
C03282=1072.363,-0.972,-62.562,172.984,23.335,154.181
C03283=1072.369,-0.722,-62.576,172.986,23.338,154.181
C03284=1072.376,-0.473,-62.590,172.987,23.340,154.181
C03285=1072.381,-0.224,-62.604,172.988,23.342,154.182
C03286=1072.387,0.026,-62.619,172.990,23.345,154.182
C03287=1072.393,0.276,-62.633,172.992,23.348,154.182
C03288=1072.398,0.525,-62.647,172.993,23.351,154.183
C03289=1072.405,0.775,-62.662,172.994,23.353,154.183
C03290=1072.410,1.024,-62.676,172.996,23.355,154.183
C03291=1072.416,1.273,-62.690,172.997,23.358,154.183
C03292=1072.422,1.524,-62.704,172.998,23.360,154.184
C03293=1072.428,1.773,-62.719,172.999,23.363,154.184
C03294=1072.433,2.022,-62.733,173.001,23.365,154.184
C03295=1072.439,2.273,-62.747,173.002,23.368,154.185
C03296=1072.446,2.521,-62.761,173.003,23.370,154.185
C03297=1072.452,2.771,-62.775,173.006,23.373,154.185
C03298=1072.458,3.020,-62.790,173.007,23.375,154.185
C03299=1072.463,3.270,-62.804,173.008,23.378,154.186
C03300=1072.470,3.520,-62.819,173.009,23.380,154.186
C03301=1072.475,3.769,-62.832,173.011,23.383,154.186
C03302=1072.481,4.018,-62.847,173.012,23.385,154.187
C03303=1072.487,4.268,-62.861,173.013,23.388,154.187
C03304=1072.493,4.517,-62.876,173.014,23.390,154.187
C03305=1072.499,4.768,-62.890,173.016,23.393,154.188
C03306=1072.505,5.017,-62.905,173.018,23.395,154.188
C03307=1072.510,5.266,-62.919,173.019,23.398,154.188
C03308=1072.516,5.516,-62.933,173.021,23.400,154.188
C03309=1072.522,5.765,-62.948,173.022,23.403,154.189
C03310=1072.528,6.015,-62.962,173.023,23.405,154.189
C03311=1072.534,6.264,-62.977,173.024,23.408,154.189
C03312=1072.540,6.514,-62.991,173.026,23.410,154.189
C03313=1072.546,6.763,-63.006,173.027,23.412,154.190
C03314=1072.552,7.014,-63.020,173.028,23.415,154.190
C03315=1072.558,7.263,-63.034,173.030,23.418,154.190
C03316=1072.564,7.511,-63.049,173.032,23.421,154.191
C03317=1072.570,7.762,-63.063,173.033,23.423,154.191
C03318=1072.575,8.011,-63.078,173.034,23.425,154.191
C03319=1072.582,8.260,-63.093,173.036,23.428,154.192
C03320=1072.587,8.510,-63.107,173.037,23.430,154.192
C03321=1072.594,8.760,-63.122,173.038,23.433,154.192
C03322=1072.600,9.009,-63.136,173.039,23.435,154.192
C03323=1072.606,9.259,-63.150,173.041,23.437,154.193
C03324=1072.611,9.508,-63.165,173.042,23.440,154.193
C03325=1072.618,9.757,-63.180,173.044,23.443,154.193
C03326=1072.623,10.007,-63.194,173.046,23.445,154.193
C03327=1072.630,10.257,-63.209,173.047,23.448,154.194
C03328=1072.635,10.506,-63.223,173.048,23.450,154.194
C03329=1072.641,10.756,-63.238,173.049,23.453,154.194
C03330=1072.647,11.005,-63.252,173.051,23.455,154.195
C03331=1072.654,11.255,-63.267,173.052,23.458,154.195
C03332=1072.659,11.503,-63.282,173.053,23.460,154.195
C03333=1072.666,11.754,-63.296,173.055,23.463,154.196
C03334=1072.672,12.003,-63.311,173.057,23.465,154.196
C03335=1072.678,12.252,-63.325,173.058,23.468,154.196
C03336=1072.684,12.502,-63.340,173.059,23.470,154.196
C03337=1072.690,12.752,-63.354,173.061,23.473,154.197
C03338=1072.696,13.001,-63.369,173.062,23.475,154.197
C03339=1072.702,13.250,-63.384,173.063,23.477,154.197
C03340=1072.708,13.500,-63.399,173.064,23.480,154.198
C03341=1072.714,13.749,-63.413,173.066,23.483,154.198
C03342=1072.720,13.999,-63.428,173.067,23.485,154.198
C03343=1072.726,14.280,-63.445,173.069,23.488,154.198
C03344=1072.734,14.560,-63.461,173.070,23.491,154.199
C03345=1072.740,14.840,-63.478,173.073,23.494,154.199
C03346=1072.747,15.121,-63.494,173.074,23.497,154.199
C03347=1072.752,15.371,-63.510,173.075,23.499,154.200
C03348=1072.758,15.620,-63.524,173.076,23.501,154.200
C03349=1072.765,15.870,-63.539,173.078,23.504,154.200
C03350=1072.770,16.119,-63.553,173.079,23.507,154.201
C03351=1072.776,16.369,-63.569,173.081,23.510,154.201
C03352=1072.782,16.618,-63.583,173.082,23.512,154.201
C03353=1072.788,16.868,-63.598,173.084,23.514,154.202
C03354=1072.794,17.117,-63.613,173.085,23.517,154.202
C03355=1072.799,17.367,-63.628,173.086,23.519,154.202
C03356=1072.806,17.616,-63.643,173.087,23.522,154.203
C03357=1072.811,17.865,-63.658,173.089,23.525,154.203
C03358=1072.818,18.115,-63.673,173.090,23.527,154.203
C03359=1072.823,18.364,-63.688,173.091,23.529,154.203
C03360=1072.829,18.614,-63.703,173.093,23.532,154.204
C03361=1072.836,18.863,-63.718,173.095,23.535,154.204
C03362=1072.841,19.113,-63.733,173.096,23.538,154.204
C03363=1072.847,19.362,-63.748,173.097,23.540,154.205
C03364=1072.853,19.611,-63.763,173.099,23.542,154.205
C03365=1072.859,19.861,-63.777,173.100,23.545,154.205
C03366=1072.865,20.111,-63.793,173.101,23.547,154.205
C03367=1072.871,20.360,-63.808,173.102,23.550,154.206
C03368=1072.877,20.610,-63.823,173.104,23.553,154.206
C03369=1072.882,20.859,-63.838,173.106,23.555,154.206
C03370=1072.889,21.108,-63.853,173.107,23.558,154.207
C03371=1072.894,21.358,-63.868,173.108,23.560,154.207
C03372=1072.900,21.607,-63.883,173.110,23.563,154.207
C03373=1072.906,21.857,-63.898,173.111,23.566,154.208
C03374=1072.912,22.107,-63.913,173.112,23.568,154.208
C03375=1072.918,22.356,-63.928,173.113,23.570,154.208
C03376=1072.923,22.606,-63.943,173.115,23.573,154.209
C03377=1072.929,22.855,-63.958,173.117,23.576,154.209
C03378=1072.935,23.105,-63.974,173.118,23.578,154.209
C03379=1072.941,23.355,-63.988,173.119,23.581,154.209
C03380=1072.947,23.604,-64.003,173.121,23.583,154.210
C03381=1072.953,23.853,-64.019,173.122,23.586,154.210
C03382=1072.959,24.103,-64.034,173.123,23.589,154.210
C03383=1072.964,24.352,-64.049,173.125,23.591,154.211
C03384=1072.971,24.601,-64.064,173.126,23.593,154.211
C03385=1072.977,24.851,-64.079,173.128,23.597,154.211
C03386=1072.982,25.100,-64.094,173.129,23.599,154.212
C03387=1072.989,25.350,-64.109,173.131,23.602,154.212
C03388=1072.995,25.599,-64.126,173.132,23.604,154.212
C03389=1073.000,25.848,-64.140,173.133,23.606,154.212
C03390=1073.006,26.098,-64.156,173.134,23.609,154.213
C03391=1073.012,26.348,-64.171,173.136,23.612,154.213
C03392=1073.018,26.598,-64.186,173.137,23.614,154.213
C03393=1073.024,26.846,-64.202,173.139,23.617,154.214
C03394=1073.030,27.096,-64.217,173.140,23.619,154.214
C03395=1073.036,27.346,-64.232,173.142,23.622,154.214
C03396=1073.041,27.595,-64.247,173.143,23.625,154.215
C03397=1073.048,27.844,-64.263,173.144,23.627,154.215
C03398=1073.053,28.094,-64.278,173.146,23.629,154.215
C03399=1073.060,28.344,-64.293,173.147,23.632,154.216
C03400=1073.065,28.593,-64.309,173.148,23.635,154.216
C03401=1073.072,28.842,-64.324,173.150,23.638,154.216
C03402=1073.077,29.092,-64.340,173.152,23.640,154.216
C03403=1073.083,29.341,-64.354,173.153,23.643,154.217
C03404=1073.089,29.590,-64.371,173.154,23.645,154.217
C03405=1073.095,29.840,-64.386,173.155,23.648,154.217
C03406=1073.101,30.090,-64.401,173.157,23.650,154.218
C03407=1073.107,30.372,-64.419,173.159,23.653,154.218
C03408=1073.114,30.654,-64.436,173.160,23.656,154.219
C03409=1073.120,30.936,-64.454,173.161,23.659,154.219
C03410=1073.128,31.217,-64.471,173.163,23.662,154.219
C03411=1073.133,31.467,-64.486,173.164,23.665,154.220
C03412=1073.139,31.716,-64.503,173.166,23.668,154.220
C03413=1073.145,31.966,-64.518,173.167,23.670,154.220
C03414=1073.151,32.216,-64.533,173.168,23.672,154.220
C03415=1073.156,32.464,-64.549,173.170,23.675,154.221
C03416=1073.162,32.714,-64.564,173.172,23.678,154.221
C03417=1073.168,32.963,-64.580,173.173,23.680,154.221
C03418=1073.174,33.213,-64.596,173.174,23.683,154.222
C03419=1073.180,33.462,-64.610,173.176,23.686,154.222
C03420=1073.186,33.711,-64.627,173.177,23.688,154.222
C03421=1073.191,33.961,-64.642,173.178,23.691,154.223
C03422=1073.198,34.210,-64.658,173.179,23.694,154.223
C03423=1073.204,34.460,-64.673,173.181,23.696,154.223
C03424=1073.209,34.709,-64.689,173.183,23.699,154.224
C03425=1073.215,34.959,-64.705,173.184,23.701,154.224
C03426=1073.221,35.208,-64.720,173.185,23.704,154.224
C03427=1073.227,35.458,-64.736,173.187,23.706,154.225
C03428=1073.233,35.707,-64.752,173.188,23.709,154.225
C03429=1073.239,35.956,-64.767,173.189,23.711,154.225
C03430=1073.245,36.206,-64.783,173.190,23.714,154.226
C03431=1073.250,36.456,-64.799,173.193,23.717,154.226
C03432=1073.257,36.705,-64.814,173.194,23.719,154.226
C03433=1073.263,36.955,-64.830,173.195,23.722,154.226
C03434=1073.269,37.204,-64.846,173.196,23.725,154.227
C03435=1073.274,37.453,-64.861,173.198,23.727,154.227
C03436=1073.280,37.702,-64.877,173.199,23.729,154.227
C03437=1073.286,37.952,-64.892,173.200,23.732,154.228
C03438=1073.292,38.202,-64.909,173.202,23.735,154.228
C03439=1073.298,38.451,-64.925,173.204,23.738,154.228
C03440=1073.303,38.701,-64.941,173.205,23.740,154.229
C03441=1073.309,38.950,-64.956,173.206,23.743,154.229
C03442=1073.315,39.199,-64.971,173.208,23.745,154.229
C03443=1073.321,39.449,-64.988,173.209,23.748,154.230
C03444=1073.327,39.698,-65.004,173.210,23.751,154.230
C03445=1073.333,39.948,-65.019,173.211,23.753,154.230
C03446=1073.339,40.197,-65.036,173.214,23.756,154.230
C03447=1073.344,40.447,-65.051,173.215,23.759,154.231
C03448=1073.350,40.696,-65.067,173.216,23.761,154.231
C03449=1073.356,40.945,-65.083,173.217,23.764,154.231
C03450=1073.361,41.195,-65.099,173.219,23.766,154.232
C03451=1073.367,41.445,-65.115,173.220,23.769,154.232
C03452=1073.374,41.694,-65.131,173.221,23.771,154.232
C03453=1073.380,41.943,-65.147,173.224,23.774,154.233
C03454=1073.385,42.192,-65.162,173.225,23.777,154.233
C03455=1073.391,42.442,-65.179,173.226,23.779,154.233
C03456=1073.397,42.691,-65.195,173.227,23.782,154.234
C03457=1073.402,42.941,-65.210,173.229,23.785,154.234
C03458=1073.408,43.190,-65.227,173.230,23.787,154.234
C03459=1073.414,43.440,-65.243,173.231,23.789,154.235
C03460=1073.420,43.689,-65.259,173.233,23.792,154.235
C03461=1073.426,43.939,-65.275,173.235,23.795,154.235
C03462=1073.432,44.188,-65.291,173.236,23.798,154.236
C03463=1073.437,44.437,-65.307,173.237,23.800,154.236
C03464=1073.443,44.686,-65.323,173.238,23.803,154.236
C03465=1073.449,44.936,-65.339,173.240,23.805,154.237
C03466=1073.455,45.186,-65.355,173.241,23.808,154.237
C03467=1073.460,45.435,-65.372,173.243,23.811,154.237
C03468=1073.466,45.685,-65.388,173.244,23.814,154.238
C03469=1073.472,45.934,-65.404,173.246,23.816,154.238
C03470=1073.478,46.183,-65.420,173.247,23.819,154.238
C03471=1073.484,46.465,-65.438,173.249,23.822,154.239
C03472=1073.491,46.747,-65.456,173.250,23.825,154.239
C03473=1073.497,47.029,-65.474,173.251,23.828,154.239
C03474=1073.504,47.311,-65.493,173.253,23.831,154.240
C03475=1073.510,47.561,-65.509,173.255,23.834,154.240
C03476=1073.514,47.810,-65.526,173.256,23.836,154.240
C03477=1073.520,48.059,-65.542,173.257,23.839,154.241
C03478=1073.526,48.308,-65.558,173.259,23.841,154.241
C03479=1073.532,48.558,-65.574,173.261,23.845,154.241
C03480=1073.538,48.807,-65.591,173.262,23.847,154.242
C03481=1073.544,49.056,-65.607,173.263,23.849,154.242
C03482=1073.549,49.306,-65.624,173.264,23.852,154.242
C03483=1073.555,49.555,-65.640,173.266,23.855,154.243
C03484=1073.561,49.805,-65.656,173.267,23.857,154.243
C03485=1073.567,50.055,-65.672,173.268,23.860,154.243
C03486=1073.573,50.304,-65.688,173.271,23.863,154.244
C03487=1073.579,50.553,-65.704,173.272,23.865,154.244
C03488=1073.584,50.803,-65.721,173.273,23.868,154.244
C03489=1073.590,51.052,-65.737,173.274,23.870,154.245
C03490=1073.596,51.302,-65.754,173.276,23.873,154.245
C03491=1073.602,51.551,-65.770,173.277,23.876,154.245
C03492=1073.608,51.800,-65.786,173.279,23.879,154.246
C03493=1073.613,52.050,-65.803,173.280,23.881,154.246
C03494=1073.619,52.299,-65.819,173.282,23.884,154.246
C03495=1073.625,52.549,-65.836,173.283,23.886,154.247
C03496=1073.631,52.797,-65.853,173.284,23.889,154.247
C03497=1073.637,53.047,-65.869,173.285,23.892,154.247
C03498=1073.642,53.296,-65.886,173.288,23.894,154.248
C03499=1073.648,53.546,-65.902,173.289,23.897,154.248
C03500=1073.654,53.795,-65.918,173.290,23.900,154.248
C03501=1073.660,54.045,-65.934,173.292,23.902,154.249
C03502=1073.666,54.294,-65.951,173.293,23.904,154.249
C03503=1073.671,54.544,-65.967,173.294,23.907,154.249
C03504=1073.677,54.793,-65.984,173.296,23.910,154.249
C03505=1073.683,55.042,-66.000,173.298,23.912,154.250
C03506=1073.689,55.292,-66.016,173.299,23.915,154.250
C03507=1073.695,55.541,-66.034,173.300,23.918,154.250
C03508=1073.701,55.790,-66.050,173.301,23.920,154.251
C03509=1073.707,56.039,-66.066,173.303,23.923,154.251
C03510=1073.713,56.289,-66.083,173.305,23.926,154.251
C03511=1073.718,56.538,-66.099,173.306,23.928,154.252
C03512=1073.724,56.788,-66.116,173.308,23.931,154.252
C03513=1073.730,57.038,-66.132,173.309,23.934,154.252
C03514=1073.737,57.286,-66.149,173.310,23.936,154.253
C03515=1073.742,57.536,-66.166,173.311,23.938,154.253
C03516=1073.748,57.785,-66.182,173.314,23.941,154.253
C03517=1073.754,58.035,-66.199,173.315,23.944,154.254
C03518=1073.760,58.284,-66.216,173.316,23.946,154.254
C03519=1073.765,58.533,-66.232,173.318,23.949,154.254
C03520=1073.771,58.783,-66.249,173.319,23.951,154.254
C03521=1073.778,59.033,-66.265,173.320,23.954,154.255
C03522=1073.783,59.282,-66.282,173.322,23.957,154.255
C03523=1073.789,59.531,-66.299,173.324,23.959,154.255
C03524=1073.795,59.780,-66.315,173.325,23.962,154.256
C03525=1073.801,60.030,-66.332,173.326,23.964,154.256
C03526=1073.807,60.279,-66.349,173.328,23.967,154.256
C03527=1073.813,60.528,-66.366,173.329,23.969,154.257
C03528=1073.819,60.778,-66.382,173.331,23.973,154.257
C03529=1073.824,61.028,-66.399,173.332,23.975,154.257
C03530=1073.831,61.277,-66.416,173.334,23.977,154.258
C03531=1073.837,61.526,-66.432,173.335,23.980,154.258
C03532=1073.842,61.776,-66.449,173.336,23.982,154.258
C03533=1073.848,62.024,-66.466,173.338,23.985,154.259
C03534=1073.855,62.274,-66.483,173.340,23.988,154.259
C03535=1073.861,62.556,-66.501,173.341,23.991,154.259
C03536=1073.868,62.838,-66.521,173.343,23.993,154.260
C03537=1073.874,63.119,-66.540,173.344,23.996,154.260
C03538=1073.882,63.401,-66.559,173.346,24.000,154.260
C03539=1073.888,63.650,-66.575,173.348,24.002,154.261
C03540=1073.893,63.900,-66.592,173.349,24.004,154.261
C03541=1073.899,64.149,-66.609,173.350,24.007,154.261
C03542=1073.905,64.398,-66.625,173.352,24.009,154.261
C03543=1073.911,64.648,-66.643,173.353,24.012,154.262
C03544=1073.916,64.897,-66.660,173.355,24.015,154.262
C03545=1073.923,65.146,-66.677,173.357,24.017,154.262
C03546=1073.928,65.396,-66.694,173.358,24.020,154.263
C03547=1073.934,65.644,-66.711,173.359,24.022,154.263
C03548=1073.940,65.895,-66.728,173.360,24.025,154.263
C03549=1073.946,66.144,-66.744,173.363,24.028,154.264
C03550=1073.951,66.393,-66.762,173.364,24.031,154.264
C03551=1073.957,66.643,-66.778,173.365,24.033,154.264
C03552=1073.963,66.892,-66.796,173.367,24.035,154.265
C03553=1073.969,67.142,-66.812,173.368,24.038,154.265
C03554=1073.975,67.391,-66.830,173.370,24.041,154.265
C03555=1073.980,67.640,-66.847,173.371,24.043,154.266
C03556=1073.986,67.889,-66.864,173.373,24.046,154.266
C03557=1073.992,68.138,-66.881,173.374,24.049,154.266
C03558=1073.998,68.388,-66.898,173.375,24.051,154.267
C03559=1074.004,68.637,-66.915,173.377,24.054,154.267
C03560=1074.010,68.887,-66.932,173.379,24.057,154.267
C03561=1074.015,69.136,-66.949,173.380,24.059,154.268
C03562=1074.021,69.386,-66.966,173.381,24.061,154.268
C03563=1074.028,69.635,-66.983,173.383,24.064,154.268
C03564=1074.033,69.884,-67.001,173.384,24.067,154.268
C03565=1074.038,70.133,-67.018,173.386,24.069,154.269
C03566=1074.045,70.382,-67.035,173.387,24.072,154.269
C03567=1074.050,70.632,-67.052,173.389,24.075,154.269
C03568=1074.056,70.881,-67.070,173.390,24.077,154.270
C03569=1074.062,71.130,-67.087,173.391,24.080,154.270
C03570=1074.067,71.380,-67.103,173.393,24.083,154.270
C03571=1074.073,71.630,-67.121,173.395,24.085,154.271
C03572=1074.079,71.879,-67.139,173.396,24.088,154.271
C03573=1074.085,72.128,-67.155,173.397,24.090,154.271
C03574=1074.090,72.377,-67.173,173.399,24.093,154.272
C03575=1074.097,72.627,-67.191,173.401,24.096,154.272
C03576=1074.103,72.876,-67.207,173.402,24.098,154.272
C03577=1074.108,73.125,-67.225,173.404,24.101,154.273
C03578=1074.114,73.375,-67.242,173.405,24.103,154.273
C03579=1074.120,73.624,-67.260,173.406,24.106,154.273
C03580=1074.125,73.874,-67.277,173.408,24.109,154.274
C03581=1074.131,74.122,-67.294,173.410,24.111,154.274
C03582=1074.137,74.372,-67.312,173.411,24.114,154.274
C03583=1074.143,74.621,-67.329,173.412,24.116,154.275
C03584=1074.148,74.871,-67.346,173.414,24.119,154.275
C03585=1074.155,75.120,-67.364,173.416,24.122,154.275
C03586=1074.160,75.369,-67.381,173.417,24.124,154.276
C03587=1074.166,75.618,-67.399,173.418,24.127,154.276
C03588=1074.172,75.868,-67.417,173.420,24.129,154.276
C03589=1074.177,76.118,-67.433,173.422,24.133,154.276
C03590=1074.183,76.366,-67.450,173.423,24.135,154.277
C03591=1074.190,76.616,-67.468,173.425,24.137,154.277
C03592=1074.195,76.865,-67.486,173.426,24.140,154.277
C03593=1074.201,77.114,-67.504,173.427,24.143,154.278
C03594=1074.208,77.364,-67.521,173.429,24.145,154.278
C03595=1074.213,77.613,-67.538,173.431,24.148,154.278
C03596=1074.218,77.862,-67.555,173.432,24.150,154.279
C03597=1074.224,78.112,-67.573,173.433,24.153,154.279
C03598=1074.230,78.361,-67.591,173.436,24.156,154.279
C03599=1074.236,78.643,-67.610,173.437,24.159,154.280
C03600=1074.243,78.924,-67.630,173.439,24.161,154.280
C03601=1074.249,79.206,-67.651,173.440,24.164,154.280
C03602=1074.255,79.487,-67.670,173.442,24.167,154.281
C03603=1074.261,79.737,-67.688,173.444,24.170,154.281
C03604=1074.267,79.986,-67.706,173.445,24.173,154.281
C03605=1074.273,80.235,-67.723,173.446,24.175,154.282
C03606=1074.279,80.485,-67.741,173.448,24.177,154.282
C03607=1074.284,80.734,-67.759,173.450,24.181,154.282
C03608=1074.290,80.983,-67.776,173.451,24.183,154.283
C03609=1074.296,81.233,-67.794,173.452,24.185,154.283
C03610=1074.301,81.482,-67.812,173.454,24.188,154.283
C03611=1074.307,81.732,-67.830,173.456,24.191,154.284
C03612=1074.313,81.981,-67.847,173.457,24.193,154.284
C03613=1074.318,82.230,-67.865,173.458,24.196,154.284
C03614=1074.325,82.479,-67.883,173.460,24.199,154.285
C03615=1074.330,82.728,-67.900,173.461,24.201,154.285
C03616=1074.336,82.977,-67.918,173.463,24.204,154.285
C03617=1074.342,83.227,-67.936,173.465,24.207,154.286
C03618=1074.347,83.476,-67.953,173.466,24.209,154.286
C03619=1074.353,83.726,-67.971,173.467,24.211,154.286
C03620=1074.359,83.975,-67.989,173.469,24.215,154.286
C03621=1074.364,84.224,-68.007,173.471,24.217,154.287
C03622=1074.371,84.474,-68.024,173.472,24.219,154.287
C03623=1074.376,84.723,-68.042,173.473,24.222,154.287
C03624=1074.382,84.973,-68.060,173.476,24.225,154.288
C03625=1074.388,85.221,-68.078,173.477,24.227,154.288
C03626=1074.394,85.471,-68.096,173.478,24.230,154.288
C03627=1074.400,85.720,-68.114,173.480,24.232,154.289
C03628=1074.406,85.970,-68.132,173.482,24.235,154.289
C03629=1074.411,86.219,-68.149,173.483,24.238,154.289
